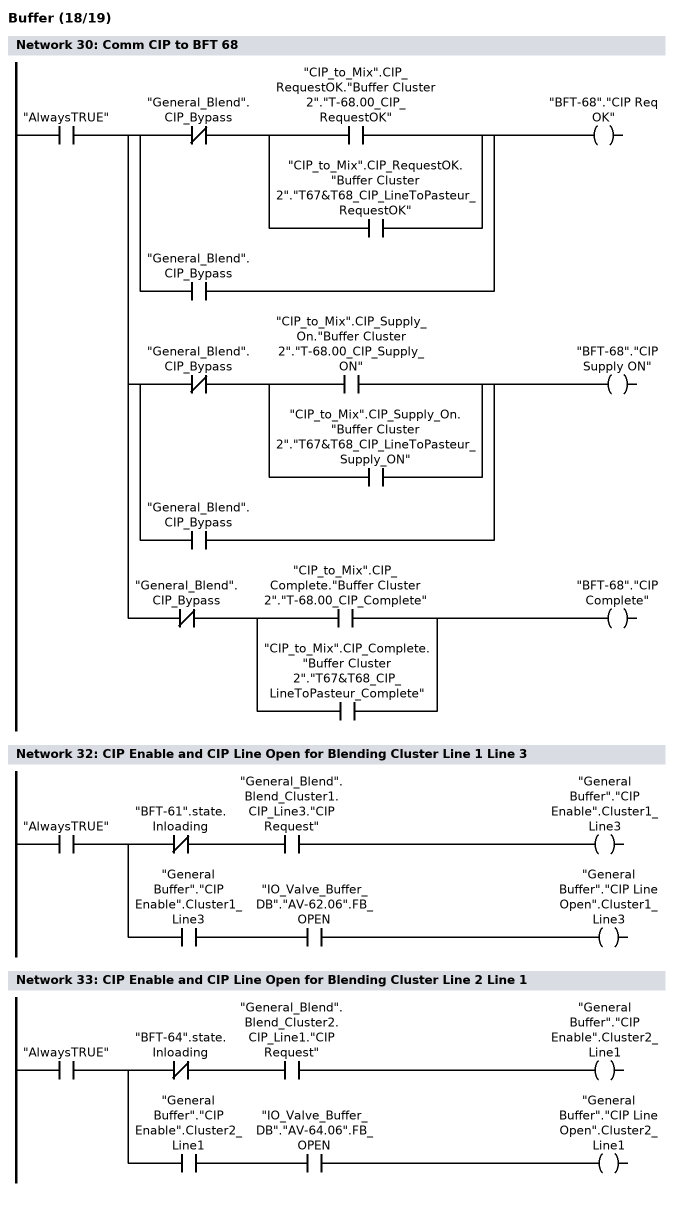
   RUNG wire#powerrail
      Contact( "AlwaysTRUE" )
      wire#w1
      I_Contact( "General_Blend".CIP_Bypass )
      wire#w2
      Contact( "CIP_to_Mix".CIP_RequestOK."Buffer Cluster 2"."T-68.00_CIP_RequestOK" )
      wire#w3
      Coil( "BFT-68"."CIP Req OK" )
   END_RUNG
   RUNG wire#w2
      Contact( "CIP_to_Mix".CIP_RequestOK."Buffer Cluster 2"."T67&T68_CIP_LineToPasteur_RequestOK" )
   END_RUNG wire#w3
   RUNG wire#w1
      Contact( "General_Blend".CIP_Bypass )
   END_RUNG wire#w3
   RUNG wire#w1
      I_Contact( "General_Blend".CIP_Bypass )
      wire#w4
      Contact( "CIP_to_Mix".CIP_Supply_On."Buffer Cluster 2"."T-68.00_CIP_Supply_ON" )
      wire#w5
      Coil( "BFT-68"."CIP Supply ON" )
   END_RUNG
   RUNG wire#w4
      Contact( "CIP_to_Mix".CIP_Supply_On."Buffer Cluster 2"."T67&T68_CIP_LineToPasteur_Supply_ON" )
   END_RUNG wire#w5
   RUNG wire#w1
      Contact( "General_Blend".CIP_Bypass )
   END_RUNG wire#w5
   RUNG wire#w1
      I_Contact( "General_Blend".CIP_Bypass )
      wire#w6
      Contact( "CIP_to_Mix".CIP_Complete."Buffer Cluster 2"."T-68.00_CIP_Complete" )
      wire#w7
      Coil( "BFT-68"."CIP Complete" )
   END_RUNG
   RUNG wire#w6
      Contact( "CIP_to_Mix".CIP_Complete."Buffer Cluster 2"."T67&T68_CIP_LineToPasteur_Complete" )
   END_RUNG wire#w7
   // the same network as SCL:
   "BFT-68"."CIP Req OK" := "AlwaysTRUE" AND ((NOT "General_Blend".CIP_Bypass AND ("CIP_to_Mix".CIP_RequestOK."Buffer Cluster 2"."T-68.00_CIP_RequestOK" OR "CIP_to_Mix".CIP_RequestOK."Buffer Cluster 2"."T67&T68_CIP_LineToPasteur_RequestOK")) OR "General_Blend".CIP_Bypass);
   "BFT-68"."CIP Supply ON" := "AlwaysTRUE" AND ((NOT "General_Blend".CIP_Bypass AND ("CIP_to_Mix".CIP_Supply_On."Buffer Cluster 2"."T-68.00_CIP_Supply_ON" OR "CIP_to_Mix".CIP_Supply_On."Buffer Cluster 2"."T67&T68_CIP_LineToPasteur_Supply_ON")) OR "General_Blend".CIP_Bypass);
   "BFT-68"."CIP Complete" := "AlwaysTRUE" AND NOT "General_Blend".CIP_Bypass AND ("CIP_to_Mix".CIP_Complete."Buffer Cluster 2"."T-68.00_CIP_Complete" OR "CIP_to_Mix".CIP_Complete."Buffer Cluster 2"."T67&T68_CIP_LineToPasteur_Complete");
END_REGION

REGION Network 32: CIP Enable and CIP Line Open for Blending Cluster Line 1 Line 3
   RUNG wire#powerrail
      Contact( "AlwaysTRUE" )
      wire#w1
      I_Contact( "BFT-61".state.Inloading )
      Contact( "General_Blend".Blend_Cluster1.CIP_Line3."CIP Request" )
      Coil( "General Buffer"."CIP Enable".Cluster1_Line3 )
   END_RUNG
   RUNG wire#w1
      Contact( "General Buffer"."CIP Enable".Cluster1_Line3 )
      Contact( "IO_Valve_Buffer_DB"."AV-62.06".FB_OPEN )
      Coil( "General Buffer"."CIP Line Open".Cluster1_Line3 )
   END_RUNG
   // the same network as SCL:
   "General Buffer"."CIP Enable".Cluster1_Line3 := "AlwaysTRUE" AND NOT "BFT-61".state.Inloading AND "General_Blend".Blend_Cluster1.CIP_Line3."CIP Request";
   "General Buffer"."CIP Line Open".Cluster1_Line3 := "AlwaysTRUE" AND "General Buffer"."CIP Enable".Cluster1_Line3 AND "IO_Valve_Buffer_DB"."AV-62.06".FB_OPEN;
END_REGION

REGION Network 33: CIP Enable and CIP Line Open for Blending Cluster Line 2 Line 1
   RUNG wire#powerrail
      Contact( "AlwaysTRUE" )
      wire#w1
      I_Contact( "BFT-64".state.Inloading )
      Contact( "General_Blend".Blend_Cluster2.CIP_Line1."CIP Request" )
      Coil( "General Buffer"."CIP Enable".Cluster2_Line1 )
   END_RUNG
   RUNG wire#w1
      Contact( "General Buffer"."CIP Enable".Cluster2_Line1 )
      Contact( "IO_Valve_Buffer_DB"."AV-64.06".FB_OPEN )
      Coil( "General Buffer"."CIP Line Open".Cluster2_Line1 )
   END_RUNG
   // the same network as SCL:
   "General Buffer"."CIP Enable".Cluster2_Line1 := "AlwaysTRUE" AND NOT "BFT-64".state.Inloading AND "General_Blend".Blend_Cluster2.CIP_Line1."CIP Request";
   "General Buffer"."CIP Line Open".Cluster2_Line1 := "AlwaysTRUE" AND "General Buffer"."CIP Enable".Cluster2_Line1 AND "IO_Valve_Buffer_DB"."AV-64.06".FB_OPEN;
END_REGION

REGION Network 34: CIP Enable and CIP Line Open for Blending Cluster Line 2 Line 2
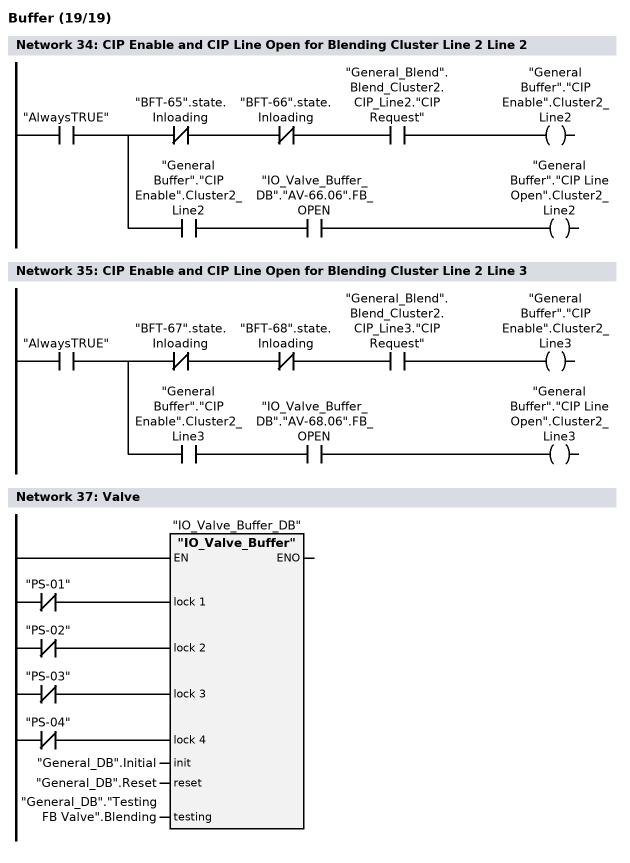
   RUNG wire#powerrail
      Contact( "AlwaysTRUE" )
      wire#w1
      I_Contact( "BFT-65".state.Inloading )
      I_Contact( "BFT-66".state.Inloading )
      Contact( "General_Blend".Blend_Cluster2.CIP_Line2."CIP Request" )
      Coil( "General Buffer"."CIP Enable".Cluster2_Line2 )
   END_RUNG
   RUNG wire#w1
      Contact( "General Buffer"."CIP Enable".Cluster2_Line2 )
      Contact( "IO_Valve_Buffer_DB"."AV-66.06".FB_OPEN )
      Coil( "General Buffer"."CIP Line Open".Cluster2_Line2 )
   END_RUNG
   // the same network as SCL:
   "General Buffer"."CIP Enable".Cluster2_Line2 := "AlwaysTRUE" AND NOT "BFT-65".state.Inloading AND NOT "BFT-66".state.Inloading AND "General_Blend".Blend_Cluster2.CIP_Line2."CIP Request";
   "General Buffer"."CIP Line Open".Cluster2_Line2 := "AlwaysTRUE" AND "General Buffer"."CIP Enable".Cluster2_Line2 AND "IO_Valve_Buffer_DB"."AV-66.06".FB_OPEN;
END_REGION

REGION Network 35: CIP Enable and CIP Line Open for Blending Cluster Line 2 Line 3
   RUNG wire#powerrail
      Contact( "AlwaysTRUE" )
      wire#w1
      I_Contact( "BFT-67".state.Inloading )
      I_Contact( "BFT-68".state.Inloading )
      Contact( "General_Blend".Blend_Cluster2.CIP_Line3."CIP Request" )
      Coil( "General Buffer"."CIP Enable".Cluster2_Line3 )
   END_RUNG
   RUNG wire#w1
      Contact( "General Buffer"."CIP Enable".Cluster2_Line3 )
      Contact( "IO_Valve_Buffer_DB"."AV-68.06".FB_OPEN )
      Coil( "General Buffer"."CIP Line Open".Cluster2_Line3 )
   END_RUNG
   // the same network as SCL:
   "General Buffer"."CIP Enable".Cluster2_Line3 := "AlwaysTRUE" AND NOT "BFT-67".state.Inloading AND NOT "BFT-68".state.Inloading AND "General_Blend".Blend_Cluster2.CIP_Line3."CIP Request";
   "General Buffer"."CIP Line Open".Cluster2_Line3 := "AlwaysTRUE" AND "General Buffer"."CIP Enable".Cluster2_Line3 AND "IO_Valve_Buffer_DB"."AV-68.06".FB_OPEN;
END_REGION

REGION Network 37: Valve
   RUNG wire#powerrail
      "IO_Valve_Buffer_DB"("lock 1" := wire#w1, "lock 2" := wire#w2, "lock 3" := wire#w3, "lock 4" := wire#w4, init := "General_DB".Initial, reset := "General_DB".Reset, testing := "General_DB"."Testing FB Valve".Blending)
   END_RUNG
   RUNG wire#powerrail
      I_Contact( "PS-01" )
   END_RUNG wire#w1
   RUNG wire#powerrail
      I_Contact( "PS-02" )
   END_RUNG wire#w2
   RUNG wire#powerrail
      I_Contact( "PS-03" )
   END_RUNG wire#w3
   RUNG wire#powerrail
      I_Contact( "PS-04" )
   END_RUNG wire#w4
   // the same network as SCL:
   "IO_Valve_Buffer_DB"("lock 1" := NOT "PS-01",   // "IO_Valve_Buffer"
                        "lock 2" := NOT "PS-02",
                        "lock 3" := NOT "PS-03",
                        "lock 4" := NOT "PS-04",
                        init := "General_DB".Initial,
                        reset := "General_DB".Reset,
                        testing := "General_DB"."Testing FB Valve".Blending);
END_REGION
END_FUNCTION

FUNCTION_BLOCK "Buffer_Tank"   // FB110, LAD
{ S7_Optimized_Access := 'TRUE' }
VERSION : 0.1
// stored: AutoNumber false, IsIECCheckEnabled false, IsRetainMemResEnabled false, MemoryReserve 100, SetENOAutomatically false, UDAEnableTagReadback false
   VAR_INPUT
      IN_LT01 : Real;
      "Tank w Circulation" : Bool;
      AlarmProd_pasteur : Bool;
      HighLevel_pasteur : Bool;
      IN_FBAV_Inload : Bool;
      IN_FBAV_CIP_Tank : Bool;
      IN_FBAV_CIP_Line : Bool;
      IN_FBAV_Outlet : Bool;
      IN_FBAV_Transfer : Bool;
      IN_FBP_Transfer : Bool;
      IN_FBXA : Bool;
      IN_FBP_Circulation : Bool;
      IN_Product_Ready : Bool;
      IN_Product_TransferOnProg : Bool;
      "Inload Busy" : Bool;
      "CIP Pulse" : Bool;
      "CIP Req OK" : Bool;
      "CIP Supply ON" : Bool;
      "CIP In Progress" : Bool;
      "CIP Complete" : Bool;
      "CIP Busy" : Bool;
   END_VAR
   VAR_OUTPUT
      Out_AV_Inload : Bool;
      Out_AV_Drain_In : Bool;
      Out_AV_CIP_Tank : Bool;
      Out_AV_CIP_Line : Bool;
      Out_AV_Outlet : Bool;
      Out_AV_Transfer : Bool;
      Out_P_Transfer : Bool;
      Out_P_Transfer_SP : Real;
      Out_XA : Bool;
      Out_XA_SP : Real;
      Out_P_Circulation : Bool;
      Out_Prod_Req : Bool;
      Out_Prod_LineOpen : Bool;
      Out_CIP_Tank_Req : Bool;
      Out_CIP_Line_Req : Bool;
      Out_CIP_Tank_LineOpen : Bool;
      Out_CIP_Line_LineOpen : Bool;
   END_VAR
   VAR
      cmd : Struct
         Inload : Bool;
         Drain_In : Bool;
         Ready_for_Transfer : Bool;
         CIP_Tank : Bool;
         CIP_Line : Bool;
         Agitator_Mode : Bool;
         Agitator_Man_OnOff : Bool;
         Agitator_SpeedMode : Bool;
         Circulation : Bool;
      END_STRUCT;
   END_VAR
   VAR RETAIN
      param : Struct
         L_Lo_Lim : Real;
         L_Hi_Lim : Real := 100.0;
         L_Hys : Real := 2.0;
         "Circulation Level" : Real := 20.0;
         SP_Level_HL : Real := 100.0;
         SP_Level_ML : Real := 80.0;
         SP_Level_LL : Real := 10.0;
         DrainIn : DInt := 10;
         SP_Pump_Transfer : Real := 80.0;
         SP_Pump_CIP : Real := 80.0;
         SP_Agitator : Real := 50.0;
         SP_Level_Agi_ON1 : Real := 20.0;
         SP_Level_Agi_OFF1 : Real := 49.0;
         SP_Level_Agi_ON2 : Real := 50.0;
         SP_Level_Agi_OFF2 : Real := 64.0;
         SP_Level_Agi_ON3 : Real := 65.0;
         "CIP Ret On" : Real := 5.0;
         "CIP Ret Off" : Real;
      END_STRUCT;
   END_VAR
   VAR
      state : Struct
         "Tank LL" : Bool;
         "Tank ML" : Bool;
         "Tank HL" : Bool;
         "Tank CIP En" : Bool;
         "Tank CIP" : Bool;
         "Line CIP En" : Bool;
         "Line CIP" : Bool;
         "Ready for Transfer En" : Bool;
         "Ready for Transfer" : Bool;
         Inloading : Bool;
         "Inload En" : Bool;
         L_Agi_ON1 : Bool;
         L_Agi_ON2 : Bool;
         L_Agi_ON3 : Bool;
         Tank_Circulation : Bool;
         "Circulation Enable" : Bool;
         Circulation : Bool;
         "Transfer on Prog" : Bool;
         "CIP Return On" : Bool;
         "CIP Req" : Bool;
      END_STRUCT;
      alwaysOn : Bool;
      L_Hys_Abs : Real;
      Hys_Level_LL : Real;
      Hys_Level_ML : Real;
      Hys_Level_HL : Real;
      Hys_Level_Circ : Real;
   END_VAR
   VAR DB_SPECIFIC
      r : Struct
         PosE1 : Bool;
         PosE2 : Bool;
         PosE3 : Bool;
         PosE4 : Bool;
         PosE5 : Bool;
         PosE6 : Bool;
         PosE7 : Bool;
         PosE8 : Bool;
         PosE9 : Bool;
         PosE10 : Bool;
         PosE11 : Bool;
         PosE12 : Bool;
         PosE13 : Bool;
         PosE14 : Bool;
         PosE15 : Bool;
         PosE16 : Bool;
         PosE17 : Bool;
         PosE18 : Bool;
         PosE19 : Bool;
         PosE20 : Bool;
         PosE21 : Bool;
         PosE22 : Bool;
         PosE23 : Bool;
         PosE24 : Bool;
         PosE25 : Bool;
         PosE26 : Bool;
         PosE27 : Bool;
         PosE28 : Bool;
         PosE29 : Bool;
         PosE30 : Bool;
         PosE31 : Bool;
         PosE32 : Bool;
      END_STRUCT;
      Actuator : Struct
         AV_Inload : Bool;
         AV_Drain_In : Bool;
         AV_Outlet : Bool;
         AV_Transfer : Bool;
         AV_CIP_Tank : Bool;
         AV_CIP_Line : Bool;
         P_Transfer : Bool;
         P_CIP : Bool;
         Agitator_level : Bool;
      END_STRUCT;
   END_VAR
   VAR
      DrainIn_OnTime : TON_TIME;
      DrainIn_OffTime : TOF_TIME;
      InloadAV_OffTime : TOF_TIME;
      DrainIn_MS : DInt;
      L_AgiTim : TON_TIME;
   END_VAR
   VAR_TEMP   // added for the SCL form of the ladder/FBD networks
      _w1 : Bool;
      _w2 : Bool;
      _w3 : Bool;
   END_VAR
BEGIN

REGION Network 1: always On
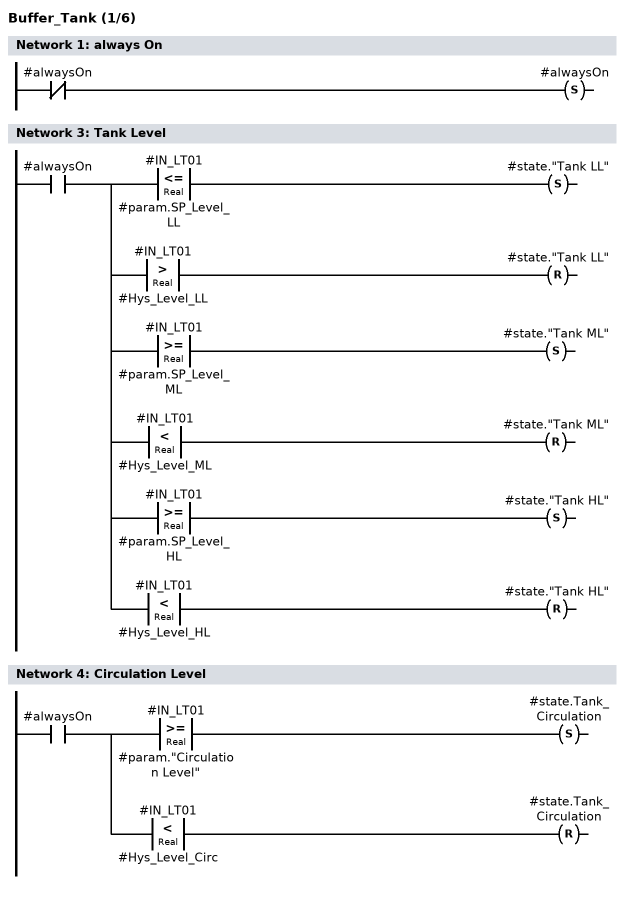
   RUNG wire#powerrail
      I_Contact( #alwaysOn )
      S_Coil( #alwaysOn )
   END_RUNG
   // the same network as SCL:
   IF NOT #alwaysOn THEN #alwaysOn := TRUE; END_IF;
END_REGION

NETWORK
TITLE = Hys Calculation
//Level Hys Absolute
      L     #param.L_Hi_Lim;
      L     #param.L_Lo_Lim;
      -R;
      L     100.0;
      /R;
      L     #param.L_Hys;
      *R;
      T     #L_Hys_Abs;
//Tank High Level
      L     #param.SP_Level_HL;
      L     #L_Hys_Abs;
      -R;
      T     #Hys_Level_HL;
//Tank Mid Level
      L     #param.SP_Level_ML;
      L     #L_Hys_Abs;
      -R;
      T     #Hys_Level_ML;
//Tank Low Level
      L     #param.SP_Level_LL;
      L     #L_Hys_Abs;
      +R;
      T     #Hys_Level_LL;
//Level Circulation
      L     #param."Circulation Level";
      L     #L_Hys_Abs;
      -R;
      T     #Hys_Level_Circ;



REGION Network 3: Tank Level
   RUNG wire#powerrail
      Contact( #alwaysOn )
      wire#w1
      { S7_Templates := "SrcType := Real" } LE_Contact(in1 := #IN_LT01, in2 := #param.SP_Level_LL)
      S_Coil( #state."Tank LL" )
   END_RUNG
   RUNG wire#w1
      { S7_Templates := "SrcType := Real" } GT_Contact(in1 := #IN_LT01, in2 := #Hys_Level_LL)
      R_Coil( #state."Tank LL" )
   END_RUNG
   RUNG wire#w1
      { S7_Templates := "SrcType := Real" } GE_Contact(in1 := #IN_LT01, in2 := #param.SP_Level_ML)
      S_Coil( #state."Tank ML" )
   END_RUNG
   RUNG wire#w1
      { S7_Templates := "SrcType := Real" } LT_Contact(in1 := #IN_LT01, in2 := #Hys_Level_ML)
      R_Coil( #state."Tank ML" )
   END_RUNG
   RUNG wire#w1
      { S7_Templates := "SrcType := Real" } GE_Contact(in1 := #IN_LT01, in2 := #param.SP_Level_HL)
      S_Coil( #state."Tank HL" )
   END_RUNG
   RUNG wire#w1
      { S7_Templates := "SrcType := Real" } LT_Contact(in1 := #IN_LT01, in2 := #Hys_Level_HL)
      R_Coil( #state."Tank HL" )
   END_RUNG
   // the same network as SCL:
   IF #alwaysOn AND (#IN_LT01 <= #param.SP_Level_LL) THEN #state."Tank LL" := TRUE; END_IF;
   IF #alwaysOn AND (#IN_LT01 > #Hys_Level_LL) THEN #state."Tank LL" := FALSE; END_IF;
   IF #alwaysOn AND (#IN_LT01 >= #param.SP_Level_ML) THEN #state."Tank ML" := TRUE; END_IF;
   IF #alwaysOn AND (#IN_LT01 < #Hys_Level_ML) THEN #state."Tank ML" := FALSE; END_IF;
   IF #alwaysOn AND (#IN_LT01 >= #param.SP_Level_HL) THEN #state."Tank HL" := TRUE; END_IF;
   IF #alwaysOn AND (#IN_LT01 < #Hys_Level_HL) THEN #state."Tank HL" := FALSE; END_IF;
END_REGION

REGION Network 4: Circulation Level
   RUNG wire#powerrail
      Contact( #alwaysOn )
      wire#w1
      { S7_Templates := "SrcType := Real" } GE_Contact(in1 := #IN_LT01, in2 := #param."Circulation Level")
      S_Coil( #state.Tank_Circulation )
   END_RUNG
   RUNG wire#w1
      { S7_Templates := "SrcType := Real" } LT_Contact(in1 := #IN_LT01, in2 := #Hys_Level_Circ)
      R_Coil( #state.Tank_Circulation )
   END_RUNG
   // the same network as SCL:
   IF #alwaysOn AND (#IN_LT01 >= #param."Circulation Level") THEN #state.Tank_Circulation := TRUE; END_IF;
   IF #alwaysOn AND (#IN_LT01 < #Hys_Level_Circ) THEN #state.Tank_Circulation := FALSE; END_IF;
END_REGION

REGION Network 5: Agitator Level ON-OFF
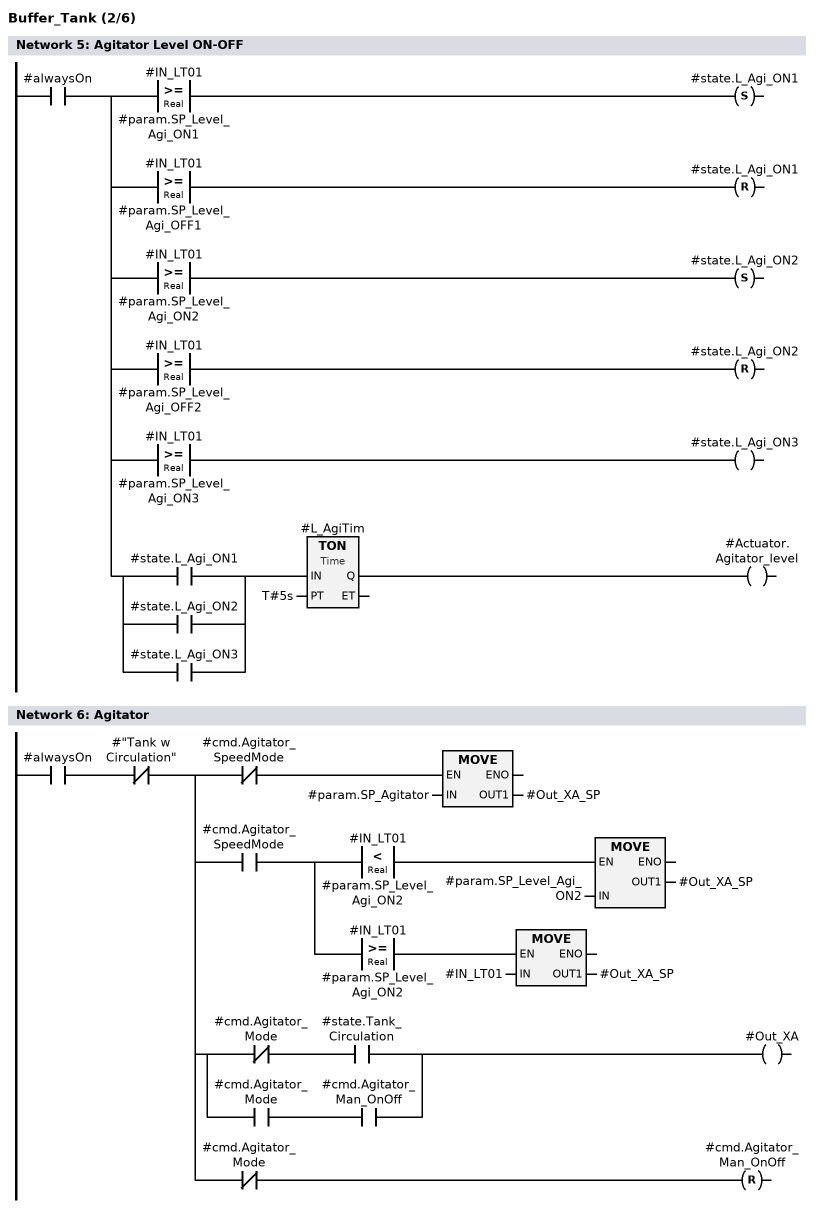
   RUNG wire#powerrail
      Contact( #alwaysOn )
      wire#w1
      { S7_Templates := "SrcType := Real" } GE_Contact(in1 := #IN_LT01, in2 := #param.SP_Level_Agi_ON1)
      S_Coil( #state.L_Agi_ON1 )
   END_RUNG
   RUNG wire#w1
      { S7_Templates := "SrcType := Real" } GE_Contact(in1 := #IN_LT01, in2 := #param.SP_Level_Agi_OFF1)
      R_Coil( #state.L_Agi_ON1 )
   END_RUNG
   RUNG wire#w1
      { S7_Templates := "SrcType := Real" } GE_Contact(in1 := #IN_LT01, in2 := #param.SP_Level_Agi_ON2)
      S_Coil( #state.L_Agi_ON2 )
   END_RUNG
   RUNG wire#w1
      { S7_Templates := "SrcType := Real" } GE_Contact(in1 := #IN_LT01, in2 := #param.SP_Level_Agi_OFF2)
      R_Coil( #state.L_Agi_ON2 )
   END_RUNG
   RUNG wire#w1
      { S7_Templates := "SrcType := Real" } GE_Contact(in1 := #IN_LT01, in2 := #param.SP_Level_Agi_ON3)
      Coil( #state.L_Agi_ON3 )
   END_RUNG
   RUNG wire#w1
      Contact( #state.L_Agi_ON1 )
      wire#w2
      { S7_Templates := "time_type := Time" } #L_AgiTim.TON(pt := T#5s, et =>)
      Coil( #Actuator.Agitator_level )
   END_RUNG
   RUNG wire#w1
      Contact( #state.L_Agi_ON2 )
   END_RUNG wire#w2
   RUNG wire#w1
      Contact( #state.L_Agi_ON3 )
   END_RUNG wire#w2
   // the same network as SCL:
   IF #alwaysOn AND (#IN_LT01 >= #param.SP_Level_Agi_ON1) THEN #state.L_Agi_ON1 := TRUE; END_IF;
   IF #alwaysOn AND (#IN_LT01 >= #param.SP_Level_Agi_OFF1) THEN #state.L_Agi_ON1 := FALSE; END_IF;
   IF #alwaysOn AND (#IN_LT01 >= #param.SP_Level_Agi_ON2) THEN #state.L_Agi_ON2 := TRUE; END_IF;
   IF #alwaysOn AND (#IN_LT01 >= #param.SP_Level_Agi_OFF2) THEN #state.L_Agi_ON2 := FALSE; END_IF;
   #state.L_Agi_ON3 := #alwaysOn AND (#IN_LT01 >= #param.SP_Level_Agi_ON3);
   #L_AgiTim(IN := #alwaysOn AND (#state.L_Agi_ON1 OR #state.L_Agi_ON2 OR #state.L_Agi_ON3), PT := T#5s);   // TON
   #Actuator.Agitator_level := #L_AgiTim.Q;
END_REGION

REGION Network 6: Agitator
   RUNG wire#powerrail
      Contact( #alwaysOn )
      I_Contact( #"Tank w Circulation" )
      wire#w1
      I_Contact( #cmd.Agitator_SpeedMode )
      Move(in := #param.SP_Agitator, out1 => #Out_XA_SP)
   END_RUNG
   RUNG wire#w1
      Contact( #cmd.Agitator_SpeedMode )
      wire#w2
      { S7_Templates := "SrcType := Real" } LT_Contact(in1 := #IN_LT01, in2 := #param.SP_Level_Agi_ON2)
      Move(in := #param.SP_Level_Agi_ON2, out1 => #Out_XA_SP)
   END_RUNG
   RUNG wire#w2
      { S7_Templates := "SrcType := Real" } GE_Contact(in1 := #IN_LT01, in2 := #param.SP_Level_Agi_ON2)
      Move(in := #IN_LT01, out1 => #Out_XA_SP)
   END_RUNG
   RUNG wire#w1
      I_Contact( #cmd.Agitator_Mode )
      Contact( #state.Tank_Circulation )
      wire#w3
      Coil( #Out_XA )
   END_RUNG
   RUNG wire#w1
      Contact( #cmd.Agitator_Mode )
      Contact( #cmd.Agitator_Man_OnOff )
   END_RUNG wire#w3
   RUNG wire#w1
      I_Contact( #cmd.Agitator_Mode )
      R_Coil( #cmd.Agitator_Man_OnOff )
   END_RUNG
   // the same network as SCL:
   #_w1 := #alwaysOn AND NOT #"Tank w Circulation";
   IF #_w1 AND NOT #cmd.Agitator_SpeedMode THEN #Out_XA_SP := #param.SP_Agitator; END_IF;
   #_w2 := #_w1 AND #cmd.Agitator_SpeedMode;
   IF #_w2 AND (#IN_LT01 < #param.SP_Level_Agi_ON2) THEN #Out_XA_SP := #param.SP_Level_Agi_ON2; END_IF;
   IF #_w2 AND (#IN_LT01 >= #param.SP_Level_Agi_ON2) THEN #Out_XA_SP := #IN_LT01; END_IF;
   #Out_XA := #_w1 AND ((NOT #cmd.Agitator_Mode AND #state.Tank_Circulation) OR (#cmd.Agitator_Mode AND #cmd.Agitator_Man_OnOff));
   IF #_w1 AND NOT #cmd.Agitator_Mode THEN #cmd.Agitator_Man_OnOff := FALSE; END_IF;
END_REGION

REGION Network 7: Circulation
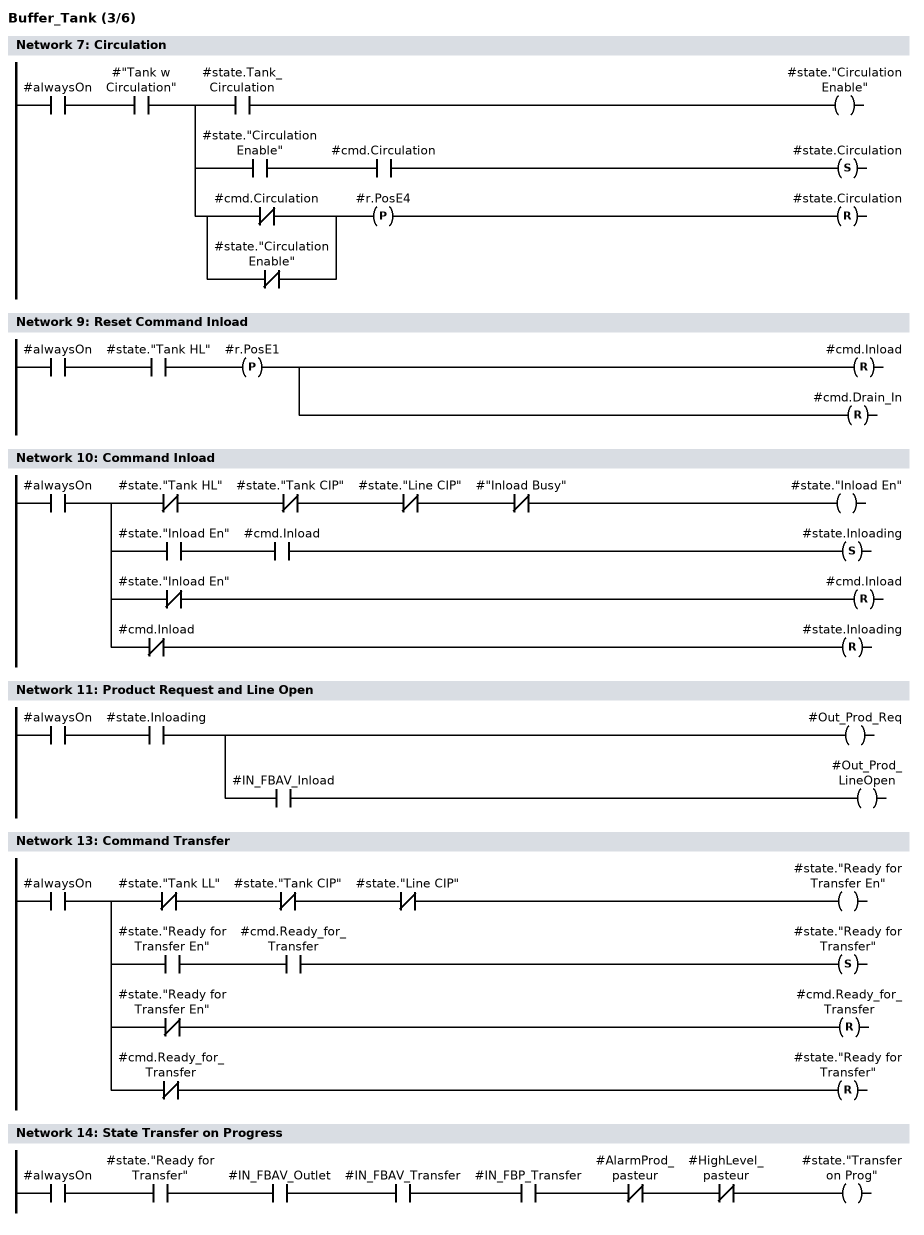
   RUNG wire#powerrail
      Contact( #alwaysOn )
      Contact( #"Tank w Circulation" )
      wire#w1
      Contact( #state.Tank_Circulation )
      Coil( #state."Circulation Enable" )
   END_RUNG
   RUNG wire#w1
      Contact( #state."Circulation Enable" )
      Contact( #cmd.Circulation )
      S_Coil( #state.Circulation )
   END_RUNG
   RUNG wire#w1
      I_Contact( #cmd.Circulation )
      wire#w2
      P_Trig( #r.PosE4 )
      R_Coil( #state.Circulation )
   END_RUNG
   RUNG wire#w1
      I_Contact( #state."Circulation Enable" )
   END_RUNG wire#w2
   // the same network as SCL:
   #_w1 := #alwaysOn AND #"Tank w Circulation";
   #state."Circulation Enable" := #_w1 AND #state.Tank_Circulation;
   IF #_w1 AND #state."Circulation Enable" AND #cmd.Circulation THEN #state.Circulation := TRUE; END_IF;
   #_w2 := #_w1 AND (NOT #cmd.Circulation OR NOT #state."Circulation Enable");
   #_w3 := #_w2 AND NOT #r.PosE4;   // rising edge
   #r.PosE4 := #_w2;
   IF #_w3 THEN #state.Circulation := FALSE; END_IF;
END_REGION

REGION Network 9: Reset Command Inload
   RUNG wire#powerrail
      Contact( #alwaysOn )
      Contact( #state."Tank HL" )
      P_Trig( #r.PosE1 )
      wire#w1
      R_Coil( #cmd.Inload )
   END_RUNG
   RUNG wire#w1
      R_Coil( #cmd.Drain_In )
   END_RUNG
   // the same network as SCL:
   #_w1 := #alwaysOn AND #state."Tank HL";
   #_w2 := #_w1 AND NOT #r.PosE1;   // rising edge
   #r.PosE1 := #_w1;
   IF #_w2 THEN
       #cmd.Inload := FALSE;
       #cmd.Drain_In := FALSE;
   END_IF;
END_REGION

REGION Network 10: Command Inload
   RUNG wire#powerrail
      Contact( #alwaysOn )
      wire#w1
      I_Contact( #state."Tank HL" )
      I_Contact( #state."Tank CIP" )
      I_Contact( #state."Line CIP" )
      I_Contact( #"Inload Busy" )
      Coil( #state."Inload En" )
   END_RUNG
   RUNG wire#w1
      Contact( #state."Inload En" )
      Contact( #cmd.Inload )
      S_Coil( #state.Inloading )
   END_RUNG
   RUNG wire#w1
      I_Contact( #state."Inload En" )
      R_Coil( #cmd.Inload )
   END_RUNG
   RUNG wire#w1
      I_Contact( #cmd.Inload )
      R_Coil( #state.Inloading )
   END_RUNG
   // the same network as SCL:
   #state."Inload En" := #alwaysOn AND NOT #state."Tank HL" AND NOT #state."Tank CIP" AND NOT #state."Line CIP" AND NOT #"Inload Busy";
   IF #alwaysOn AND #state."Inload En" AND #cmd.Inload THEN #state.Inloading := TRUE; END_IF;
   IF #alwaysOn AND NOT #state."Inload En" THEN #cmd.Inload := FALSE; END_IF;
   IF #alwaysOn AND NOT #cmd.Inload THEN #state.Inloading := FALSE; END_IF;
END_REGION

REGION Network 11: Product Request and Line Open
   RUNG wire#powerrail
      Contact( #alwaysOn )
      Contact( #state.Inloading )
      wire#w1
      Coil( #Out_Prod_Req )
   END_RUNG
   RUNG wire#w1
      Contact( #IN_FBAV_Inload )
      Coil( #Out_Prod_LineOpen )
   END_RUNG
   // the same network as SCL:
   #Out_Prod_Req := #alwaysOn AND #state.Inloading;
   #Out_Prod_LineOpen := #Out_Prod_Req AND #IN_FBAV_Inload;
END_REGION

REGION Network 13: Command Transfer
   RUNG wire#powerrail
      Contact( #alwaysOn )
      wire#w1
      I_Contact( #state."Tank LL" )
      I_Contact( #state."Tank CIP" )
      I_Contact( #state."Line CIP" )
      Coil( #state."Ready for Transfer En" )
   END_RUNG
   RUNG wire#w1
      Contact( #state."Ready for Transfer En" )
      Contact( #cmd.Ready_for_Transfer )
      S_Coil( #state."Ready for Transfer" )
   END_RUNG
   RUNG wire#w1
      I_Contact( #state."Ready for Transfer En" )
      R_Coil( #cmd.Ready_for_Transfer )
   END_RUNG
   RUNG wire#w1
      I_Contact( #cmd.Ready_for_Transfer )
      R_Coil( #state."Ready for Transfer" )
   END_RUNG
   // the same network as SCL:
   #state."Ready for Transfer En" := #alwaysOn AND NOT #state."Tank LL" AND NOT #state."Tank CIP" AND NOT #state."Line CIP";
   IF #alwaysOn AND #state."Ready for Transfer En" AND #cmd.Ready_for_Transfer THEN
       #state."Ready for Transfer" := TRUE;
   END_IF;
   IF #alwaysOn AND NOT #state."Ready for Transfer En" THEN #cmd.Ready_for_Transfer := FALSE; END_IF;
   IF #alwaysOn AND NOT #cmd.Ready_for_Transfer THEN #state."Ready for Transfer" := FALSE; END_IF;
END_REGION

REGION Network 14: State Transfer on Progress
   RUNG wire#powerrail
      Contact( #alwaysOn )
      Contact( #state."Ready for Transfer" )
      Contact( #IN_FBAV_Outlet )
      Contact( #IN_FBAV_Transfer )
      Contact( #IN_FBP_Transfer )
      I_Contact( #AlarmProd_pasteur )
      I_Contact( #HighLevel_pasteur )
      Coil( #state."Transfer on Prog" )
   END_RUNG
   // the same network as SCL:
   #state."Transfer on Prog" := #alwaysOn AND #state."Ready for Transfer" AND #IN_FBAV_Outlet AND #IN_FBAV_Transfer AND #IN_FBP_Transfer AND NOT #AlarmProd_pasteur AND NOT #HighLevel_pasteur;
END_REGION

REGION Network 16: Command CIP
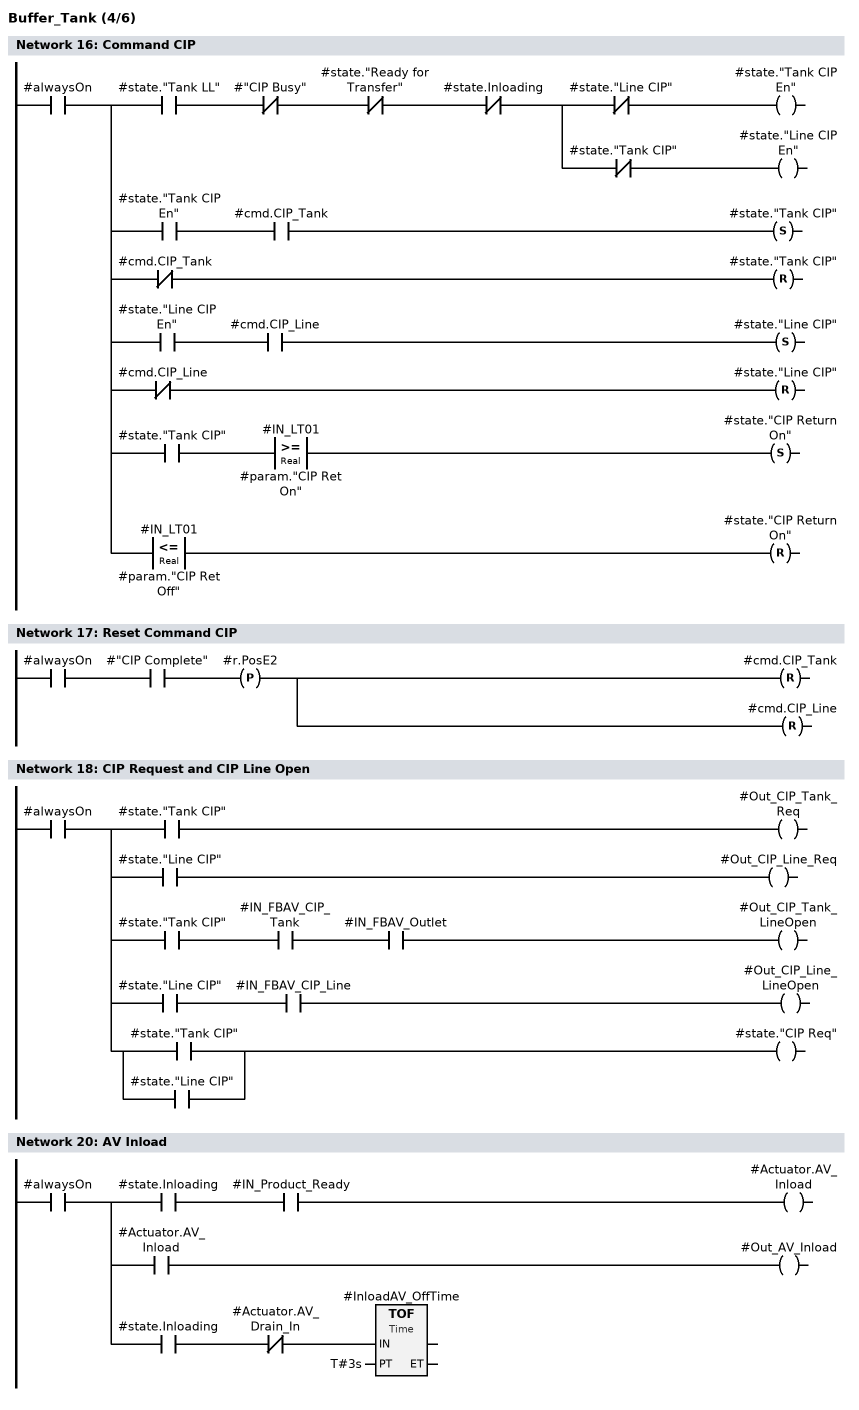
   RUNG wire#powerrail
      Contact( #alwaysOn )
      wire#w1
      Contact( #state."Tank LL" )
      I_Contact( #"CIP Busy" )
      I_Contact( #state."Ready for Transfer" )
      I_Contact( #state.Inloading )
      wire#w2
      I_Contact( #state."Line CIP" )
      Coil( #state."Tank CIP En" )
   END_RUNG
   RUNG wire#w2
      I_Contact( #state."Tank CIP" )
      Coil( #state."Line CIP En" )
   END_RUNG
   RUNG wire#w1
      Contact( #state."Tank CIP En" )
      Contact( #cmd.CIP_Tank )
      S_Coil( #state."Tank CIP" )
   END_RUNG
   RUNG wire#w1
      I_Contact( #cmd.CIP_Tank )
      R_Coil( #state."Tank CIP" )
   END_RUNG
   RUNG wire#w1
      Contact( #state."Line CIP En" )
      Contact( #cmd.CIP_Line )
      S_Coil( #state."Line CIP" )
   END_RUNG
   RUNG wire#w1
      I_Contact( #cmd.CIP_Line )
      R_Coil( #state."Line CIP" )
   END_RUNG
   RUNG wire#w1
      Contact( #state."Tank CIP" )
      { S7_Templates := "SrcType := Real" } GE_Contact(in1 := #IN_LT01, in2 := #param."CIP Ret On")
      S_Coil( #state."CIP Return On" )
   END_RUNG
   RUNG wire#w1
      { S7_Templates := "SrcType := Real" } LE_Contact(in1 := #IN_LT01, in2 := #param."CIP Ret Off")
      R_Coil( #state."CIP Return On" )
   END_RUNG
   // the same network as SCL:
   #_w1 := #alwaysOn AND #state."Tank LL" AND NOT #"CIP Busy" AND NOT #state."Ready for Transfer" AND NOT #state.Inloading;
   #state."Tank CIP En" := #_w1 AND NOT #state."Line CIP";
   #state."Line CIP En" := #_w1 AND NOT #state."Tank CIP";
   IF #alwaysOn AND #state."Tank CIP En" AND #cmd.CIP_Tank THEN #state."Tank CIP" := TRUE; END_IF;
   IF #alwaysOn AND NOT #cmd.CIP_Tank THEN #state."Tank CIP" := FALSE; END_IF;
   IF #alwaysOn AND #state."Line CIP En" AND #cmd.CIP_Line THEN #state."Line CIP" := TRUE; END_IF;
   IF #alwaysOn AND NOT #cmd.CIP_Line THEN #state."Line CIP" := FALSE; END_IF;
   IF #alwaysOn AND #state."Tank CIP" AND (#IN_LT01 >= #param."CIP Ret On") THEN
       #state."CIP Return On" := TRUE;
   END_IF;
   IF #alwaysOn AND (#IN_LT01 <= #param."CIP Ret Off") THEN #state."CIP Return On" := FALSE; END_IF;
END_REGION

REGION Network 17: Reset Command CIP
   RUNG wire#powerrail
      Contact( #alwaysOn )
      Contact( #"CIP Complete" )
      P_Trig( #r.PosE2 )
      wire#w1
      R_Coil( #cmd.CIP_Tank )
   END_RUNG
   RUNG wire#w1
      R_Coil( #cmd.CIP_Line )
   END_RUNG
   // the same network as SCL:
   #_w1 := #alwaysOn AND #"CIP Complete";
   #_w2 := #_w1 AND NOT #r.PosE2;   // rising edge
   #r.PosE2 := #_w1;
   IF #_w2 THEN
       #cmd.CIP_Tank := FALSE;
       #cmd.CIP_Line := FALSE;
   END_IF;
END_REGION

REGION Network 18: CIP Request and CIP Line Open
   RUNG wire#powerrail
      Contact( #alwaysOn )
      wire#w1
      Contact( #state."Tank CIP" )
      Coil( #Out_CIP_Tank_Req )
   END_RUNG
   RUNG wire#w1
      Contact( #state."Line CIP" )
      Coil( #Out_CIP_Line_Req )
   END_RUNG
   RUNG wire#w1
      Contact( #state."Tank CIP" )
      Contact( #IN_FBAV_CIP_Tank )
      Contact( #IN_FBAV_Outlet )
      Coil( #Out_CIP_Tank_LineOpen )
   END_RUNG
   RUNG wire#w1
      Contact( #state."Line CIP" )
      Contact( #IN_FBAV_CIP_Line )
      Coil( #Out_CIP_Line_LineOpen )
   END_RUNG
   RUNG wire#w1
      Contact( #state."Tank CIP" )
      wire#w2
      Coil( #state."CIP Req" )
   END_RUNG
   RUNG wire#w1
      Contact( #state."Line CIP" )
   END_RUNG wire#w2
   // the same network as SCL:
   #Out_CIP_Tank_Req := #alwaysOn AND #state."Tank CIP";
   #Out_CIP_Line_Req := #alwaysOn AND #state."Line CIP";
   #Out_CIP_Tank_LineOpen := #alwaysOn AND #state."Tank CIP" AND #IN_FBAV_CIP_Tank AND #IN_FBAV_Outlet;
   #Out_CIP_Line_LineOpen := #alwaysOn AND #state."Line CIP" AND #IN_FBAV_CIP_Line;
   #state."CIP Req" := #alwaysOn AND (#state."Tank CIP" OR #state."Line CIP");
END_REGION

REGION Network 20: AV Inload
   RUNG wire#powerrail
      Contact( #alwaysOn )
      wire#w1
      Contact( #state.Inloading )
      Contact( #IN_Product_Ready )
      Coil( #Actuator.AV_Inload )
   END_RUNG
   RUNG wire#w1
      Contact( #Actuator.AV_Inload )
      Coil( #Out_AV_Inload )
   END_RUNG
   RUNG wire#w1
      Contact( #state.Inloading )
      I_Contact( #Actuator.AV_Drain_In )
      { S7_Templates := "time_type := Time" } #InloadAV_OffTime.TOF(pt := T#3s, et =>)
   END_RUNG
   // the same network as SCL:
   #Actuator.AV_Inload := #alwaysOn AND #state.Inloading AND #IN_Product_Ready;
   #Out_AV_Inload := #alwaysOn AND #Actuator.AV_Inload;
   #InloadAV_OffTime(IN := #alwaysOn AND #state.Inloading AND NOT #Actuator.AV_Drain_In, PT := T#3s);   // TOF
END_REGION

REGION Network 21: AV Drain In
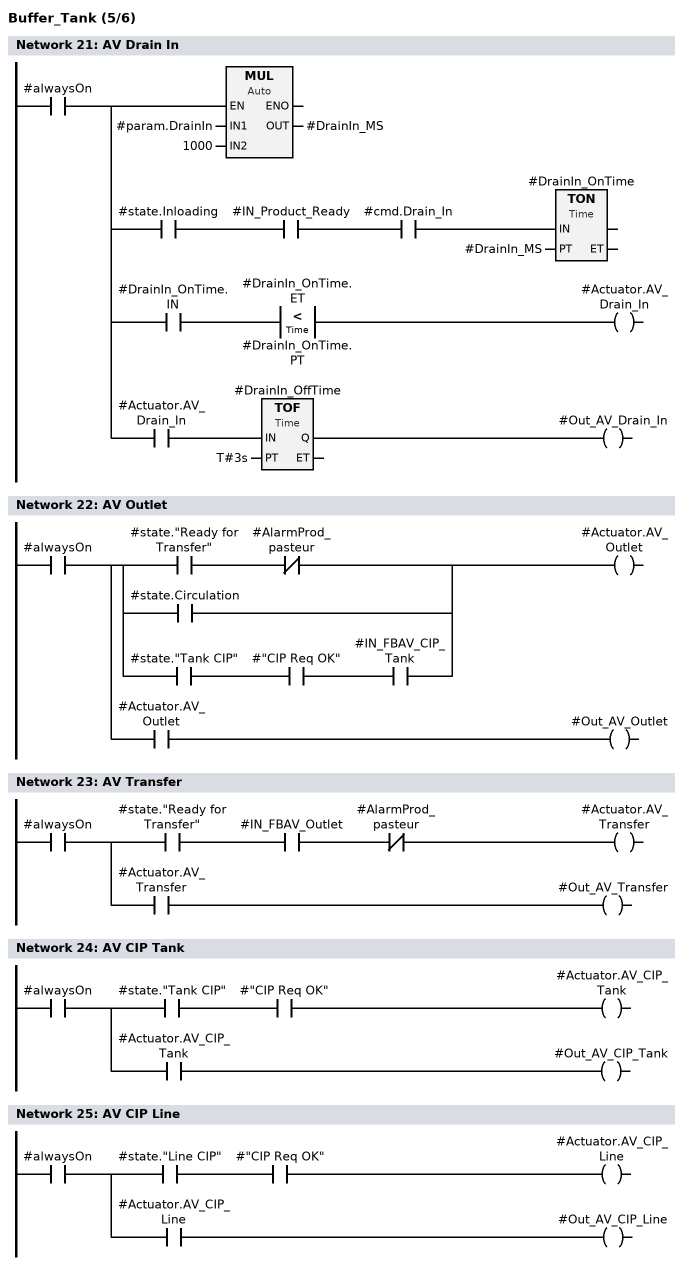
   RUNG wire#powerrail
      Contact( #alwaysOn )
      wire#w1
      Mul(in1 := #param.DrainIn, in2 := 1000, out => #DrainIn_MS)
   END_RUNG
   RUNG wire#w1
      Contact( #state.Inloading )
      Contact( #IN_Product_Ready )
      Contact( #cmd.Drain_In )
      { S7_Templates := "time_type := Time" } #DrainIn_OnTime.TON(pt := #DrainIn_MS, et =>)
   END_RUNG
   RUNG wire#w1
      Contact( #DrainIn_OnTime.IN )
      { S7_Templates := "SrcType := Time" } LT_Contact(in1 := #DrainIn_OnTime.ET, in2 := #DrainIn_OnTime.PT)
      Coil( #Actuator.AV_Drain_In )
   END_RUNG
   RUNG wire#w1
      Contact( #Actuator.AV_Drain_In )
      { S7_Templates := "time_type := Time" } #DrainIn_OffTime.TOF(pt := T#3s, et =>)
      Coil( #Out_AV_Drain_In )
   END_RUNG
   // the same network as SCL:
   IF #alwaysOn THEN #DrainIn_MS := #param.DrainIn * 1000; END_IF;
   #DrainIn_OnTime(IN := #alwaysOn AND #state.Inloading AND #IN_Product_Ready AND #cmd.Drain_In,   // TON
                   PT := #DrainIn_MS);
   #Actuator.AV_Drain_In := #alwaysOn AND #DrainIn_OnTime.IN AND (#DrainIn_OnTime.ET < #DrainIn_OnTime.PT);
   #DrainIn_OffTime(IN := #alwaysOn AND #Actuator.AV_Drain_In, PT := T#3s);   // TOF
   #Out_AV_Drain_In := #DrainIn_OffTime.Q;
END_REGION

REGION Network 22: AV Outlet
   RUNG wire#powerrail
      Contact( #alwaysOn )
      wire#w1
      Contact( #state."Ready for Transfer" )
      I_Contact( #AlarmProd_pasteur )
      wire#w2
      Coil( #Actuator.AV_Outlet )
   END_RUNG
   RUNG wire#w1
      Contact( #state.Circulation )
   END_RUNG wire#w2
   RUNG wire#w1
      Contact( #state."Tank CIP" )
      Contact( #"CIP Req OK" )
      Contact( #IN_FBAV_CIP_Tank )
   END_RUNG wire#w2
   RUNG wire#w1
      Contact( #Actuator.AV_Outlet )
      Coil( #Out_AV_Outlet )
   END_RUNG
   // the same network as SCL:
   #Actuator.AV_Outlet := #alwaysOn AND ((#state."Ready for Transfer" AND NOT #AlarmProd_pasteur) OR #state.Circulation OR (#state."Tank CIP" AND #"CIP Req OK" AND #IN_FBAV_CIP_Tank));
   #Out_AV_Outlet := #alwaysOn AND #Actuator.AV_Outlet;
END_REGION

REGION Network 23: AV Transfer
   RUNG wire#powerrail
      Contact( #alwaysOn )
      wire#w1
      Contact( #state."Ready for Transfer" )
      Contact( #IN_FBAV_Outlet )
      I_Contact( #AlarmProd_pasteur )
      Coil( #Actuator.AV_Transfer )
   END_RUNG
   RUNG wire#w1
      Contact( #Actuator.AV_Transfer )
      Coil( #Out_AV_Transfer )
   END_RUNG
   // the same network as SCL:
   #Actuator.AV_Transfer := #alwaysOn AND #state."Ready for Transfer" AND #IN_FBAV_Outlet AND NOT #AlarmProd_pasteur;
   #Out_AV_Transfer := #alwaysOn AND #Actuator.AV_Transfer;
END_REGION

REGION Network 24: AV CIP Tank
   RUNG wire#powerrail
      Contact( #alwaysOn )
      wire#w1
      Contact( #state."Tank CIP" )
      Contact( #"CIP Req OK" )
      Coil( #Actuator.AV_CIP_Tank )
   END_RUNG
   RUNG wire#w1
      Contact( #Actuator.AV_CIP_Tank )
      Coil( #Out_AV_CIP_Tank )
   END_RUNG
   // the same network as SCL:
   #Actuator.AV_CIP_Tank := #alwaysOn AND #state."Tank CIP" AND #"CIP Req OK";
   #Out_AV_CIP_Tank := #alwaysOn AND #Actuator.AV_CIP_Tank;
END_REGION

REGION Network 25: AV CIP Line
   RUNG wire#powerrail
      Contact( #alwaysOn )
      wire#w1
      Contact( #state."Line CIP" )
      Contact( #"CIP Req OK" )
      Coil( #Actuator.AV_CIP_Line )
   END_RUNG
   RUNG wire#w1
      Contact( #Actuator.AV_CIP_Line )
      Coil( #Out_AV_CIP_Line )
   END_RUNG
   // the same network as SCL:
   #Actuator.AV_CIP_Line := #alwaysOn AND #state."Line CIP" AND #"CIP Req OK";
   #Out_AV_CIP_Line := #alwaysOn AND #Actuator.AV_CIP_Line;
END_REGION

REGION Network 27: Pump Transfer
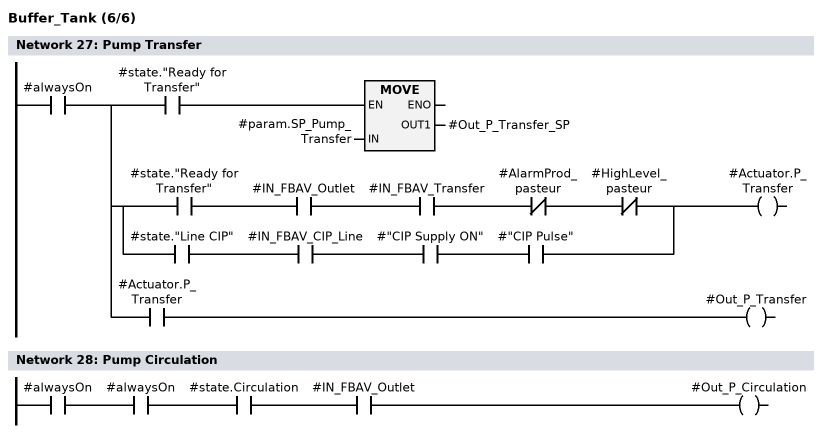
   RUNG wire#powerrail
      Contact( #alwaysOn )
      wire#w1
      Contact( #state."Ready for Transfer" )
      Move(in := #param.SP_Pump_Transfer, out1 => #Out_P_Transfer_SP)
   END_RUNG
   RUNG wire#w1
      Contact( #state."Ready for Transfer" )
      Contact( #IN_FBAV_Outlet )
      Contact( #IN_FBAV_Transfer )
      I_Contact( #AlarmProd_pasteur )
      I_Contact( #HighLevel_pasteur )
      wire#w2
      Coil( #Actuator.P_Transfer )
   END_RUNG
   RUNG wire#w1
      Contact( #state."Line CIP" )
      Contact( #IN_FBAV_CIP_Line )
      Contact( #"CIP Supply ON" )
      Contact( #"CIP Pulse" )
   END_RUNG wire#w2
   RUNG wire#w1
      Contact( #Actuator.P_Transfer )
      Coil( #Out_P_Transfer )
   END_RUNG
   // the same network as SCL:
   IF #alwaysOn AND #state."Ready for Transfer" THEN #Out_P_Transfer_SP := #param.SP_Pump_Transfer; END_IF;
   #Actuator.P_Transfer := #alwaysOn AND ((#state."Ready for Transfer" AND #IN_FBAV_Outlet AND #IN_FBAV_Transfer AND NOT #AlarmProd_pasteur AND NOT #HighLevel_pasteur) OR (#state."Line CIP" AND #IN_FBAV_CIP_Line AND #"CIP Supply ON" AND #"CIP Pulse"));
   #Out_P_Transfer := #alwaysOn AND #Actuator.P_Transfer;
END_REGION

REGION Network 28: Pump Circulation
   RUNG wire#powerrail
      Contact( #alwaysOn )
      Contact( #alwaysOn )
      Contact( #state.Circulation )
      Contact( #IN_FBAV_Outlet )
      Coil( #Out_P_Circulation )
   END_RUNG
   // the same network as SCL:
   #Out_P_Circulation := #alwaysOn AND #alwaysOn AND #state.Circulation AND #IN_FBAV_Outlet;
END_REGION
END_FUNCTION_BLOCK

FUNCTION_BLOCK "IO_Valve_Buffer"   // FB19, LAD
{ S7_Optimized_Access := 'FALSE' }
VERSION : 0.1
// stored: AutoNumber true, IsIECCheckEnabled false, SetENOAutomatically false, UDAEnableTagReadback false
   VAR_INPUT
      "lock 1" : Bool;
      "lock 2" : Bool;
      "lock 3" : Bool;
      "lock 4" : Bool;
      init : Bool;
      reset : Bool;
      testing : Bool;
   END_VAR
   VAR
      "AV-22.11" : "Valve";
      "AV-22.21" : "Valve";
      "AV-22.22" : "Valve";
      "AV-22.23" : "Valve";
      "AV-32.01" : "Valve";
      "AV-32.02" : "Valve";
      "AV-32.03" : "Valve";
      "AV-32.04" : "Valve";
      "AV-32.11" : "Valve";
      "AV-32.21" : "Valve";
      "AV-32.22" : "Valve";
      "AV-32.23" : "Valve";
      "AV-61.01" : "Valve";
      "AV-61.02" : "Valve";
      "AV-61.03" : "Valve";
      "AV-61.04" : "Valve";
      "AV-61.05" : "Valve";
      "AV-61.21" : "Valve";
      "AV-62.06" : "Valve";
      "AV-64.01" : "Valve";
      "AV-64.02" : "Valve";
      "AV-64.03" : "Valve";
      "AV-64.04" : "Valve";
      "AV-64.05" : "Valve";
      "AV-64.06" : "Valve";
      "AV-65.01" : "Valve";
      "AV-65.02" : "Valve";
      "AV-65.03" : "Valve";
      "AV-65.04" : "Valve";
      "AV-65.05" : "Valve";
      "AV-65.21" : "Valve";
      "AV-66.01" : "Valve";
      "AV-66.02" : "Valve";
      "AV-66.03" : "Valve";
      "AV-66.04" : "Valve";
      "AV-66.05" : "Valve";
      "AV-66.06" : "Valve";
      "AV-67.01" : "Valve";
      "AV-67.02" : "Valve";
      "AV-67.03" : "Valve";
      "AV-67.04" : "Valve";
      "AV-67.05" : "Valve";
      "AV-68.01" : "Valve";
      "AV-68.02" : "Valve";
      "AV-68.03" : "Valve";
      "AV-68.04" : "Valve";
      "AV-68.05" : "Valve";
      "AV-68.06" : "Valve";
   END_VAR
BEGIN

REGION Network 1 (SCL): FB OPEN AND CLOSE VALVE T-22
   IF #testing THEN
       // Statement section IF
       #"AV-22.11".FB_OPEN := #"AV-22.11".QCMD_OP;
       #"AV-22.11".FB_CLOSE := NOT #"AV-22.11".QCMD_OP;
       #"AV-22.21".FB_OPEN := #"AV-22.21".QCMD_OP;
       #"AV-22.21".FB_CLOSE := NOT #"AV-22.21".QCMD_OP;
       #"AV-22.22".FB_OPEN := #"AV-22.22".QCMD_OP;
       #"AV-22.22".FB_CLOSE := NOT #"AV-22.22".QCMD_OP;
       #"AV-22.23".FB_OPEN := #"AV-22.23".QCMD_OP;
       #"AV-22.23".FB_CLOSE := NOT #"AV-22.23".QCMD_OP;
   ELSE
       // Statement section ELSE
       #"AV-22.11".FB_OPEN := #"AV-22.11".QCMD_OP;
       #"AV-22.11".FB_CLOSE := NOT #"AV-22.11".QCMD_OP;
       #"AV-22.21".FB_OPEN := #"AV-22.21".QCMD_OP;
       #"AV-22.21".FB_CLOSE := NOT #"AV-22.21".QCMD_OP;
       #"AV-22.22".FB_OPEN := #"AV-22.22".QCMD_OP;
       #"AV-22.22".FB_CLOSE := NOT #"AV-22.22".QCMD_OP;
       #"AV-22.23".FB_OPEN := #"AV-22.23".QCMD_OP;
       #"AV-22.23".FB_CLOSE := NOT #"AV-22.23".QCMD_OP;
   END_IF;
END_REGION

NETWORK
TITLE = FB MONITORING TIME VALVE T-22
// FB OPEN TIME
      L     T#20s;
      T     #"AV-22.11".MON_T;
      T     #"AV-22.21".MON_T;
      T     #"AV-22.22".MON_T;
      T     #"AV-22.23".MON_T;
// FB CLOSE TIME
      L     T#20s;
      T     #"AV-22.11".MON_T_CLOSE;
      T     #"AV-22.21".MON_T_CLOSE;
      T     #"AV-22.22".MON_T_CLOSE;
      T     #"AV-22.23".MON_T_CLOSE;


REGION Network 3: AV-22.11
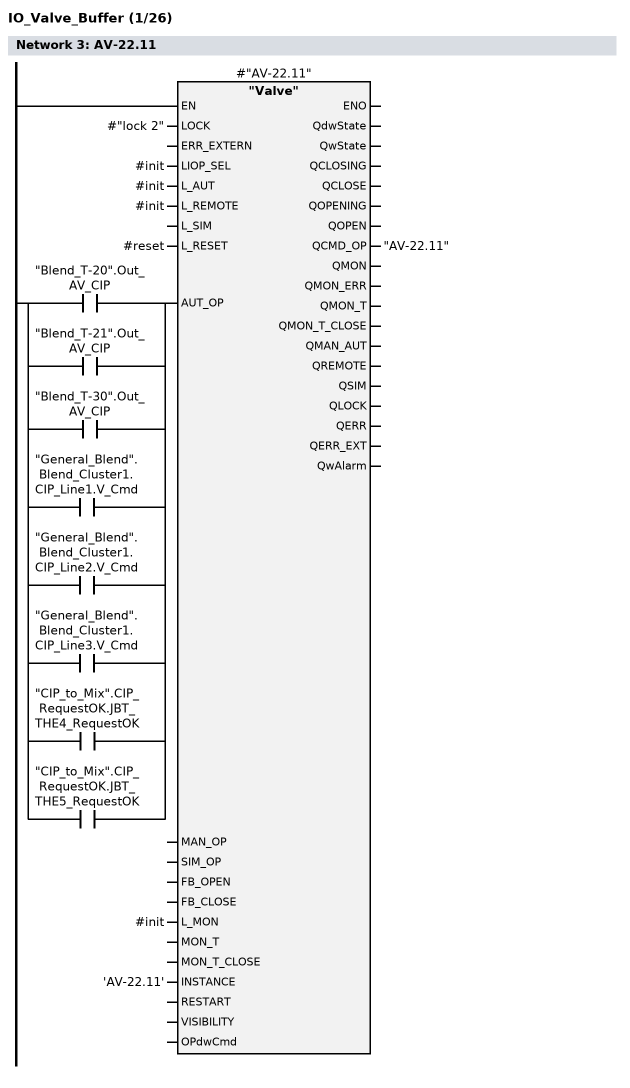
   RUNG wire#powerrail
      #"AV-22.11"(AUT_OP := wire#w1, LOCK := #"lock 2", ERR_EXTERN :=, LIOP_SEL := #init, L_AUT := #init, L_REMOTE := #init, L_SIM :=, L_RESET := #reset, MAN_OP :=, SIM_OP :=, FB_OPEN :=, FB_CLOSE :=, L_MON := #init, MON_T :=, MON_T_CLOSE :=, INSTANCE := 'AV-22.11', RESTART :=, VISIBILITY :=, OPdwCmd :=, QdwState =>, QwState =>, QCLOSING =>, QCLOSE =>, QOPENING =>, QOPEN =>, QCMD_OP => "AV-22.11", QMON =>, QMON_ERR =>, QMON_T =>, QMON_T_CLOSE =>, QMAN_AUT =>, QREMOTE =>, QSIM =>, QLOCK =>, QERR =>, QERR_EXT =>, QwAlarm =>)
   END_RUNG
   RUNG wire#powerrail
      Contact( "Blend_T-20".Out_AV_CIP )
   END_RUNG wire#w1
   RUNG wire#powerrail
      Contact( "Blend_T-21".Out_AV_CIP )
   END_RUNG wire#w1
   RUNG wire#powerrail
      Contact( "Blend_T-30".Out_AV_CIP )
   END_RUNG wire#w1
   RUNG wire#powerrail
      Contact( "General_Blend".Blend_Cluster1.CIP_Line1.V_Cmd )
   END_RUNG wire#w1
   RUNG wire#powerrail
      Contact( "General_Blend".Blend_Cluster1.CIP_Line2.V_Cmd )
   END_RUNG wire#w1
   RUNG wire#powerrail
      Contact( "General_Blend".Blend_Cluster1.CIP_Line3.V_Cmd )
   END_RUNG wire#w1
   RUNG wire#powerrail
      Contact( "CIP_to_Mix".CIP_RequestOK.JBT_THE4_RequestOK )
   END_RUNG wire#w1
   RUNG wire#powerrail
      Contact( "CIP_to_Mix".CIP_RequestOK.JBT_THE5_RequestOK )
   END_RUNG wire#w1
   // the same network as SCL:
   #"AV-22.11"(LOCK := #"lock 2",   // "Valve"
               LIOP_SEL := #init,
               L_AUT := #init,
               L_REMOTE := #init,
               L_RESET := #reset,
               AUT_OP := "Blend_T-20".Out_AV_CIP OR "Blend_T-21".Out_AV_CIP OR "Blend_T-30".Out_AV_CIP OR "General_Blend".Blend_Cluster1.CIP_Line1.V_Cmd OR "General_Blend".Blend_Cluster1.CIP_Line2.V_Cmd OR "General_Blend".Blend_Cluster1.CIP_Line3.V_Cmd OR "CIP_to_Mix".CIP_RequestOK.JBT_THE4_RequestOK OR "CIP_to_Mix".CIP_RequestOK.JBT_THE5_RequestOK,
               L_MON := #init,
               INSTANCE := 'AV-22.11',
               QCMD_OP => "AV-22.11");
END_REGION

REGION Network 4: AV-22.21
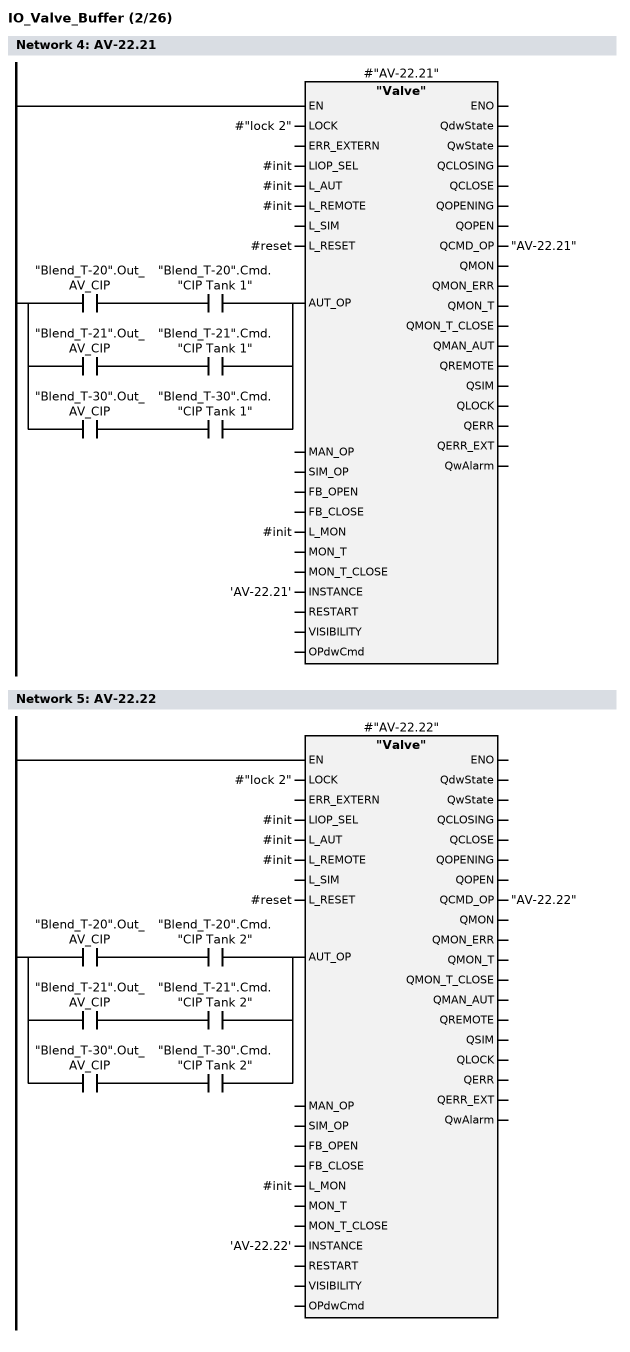
   RUNG wire#powerrail
      #"AV-22.21"(AUT_OP := wire#w1, LOCK := #"lock 2", ERR_EXTERN :=, LIOP_SEL := #init, L_AUT := #init, L_REMOTE := #init, L_SIM :=, L_RESET := #reset, MAN_OP :=, SIM_OP :=, FB_OPEN :=, FB_CLOSE :=, L_MON := #init, MON_T :=, MON_T_CLOSE :=, INSTANCE := 'AV-22.21', RESTART :=, VISIBILITY :=, OPdwCmd :=, QdwState =>, QwState =>, QCLOSING =>, QCLOSE =>, QOPENING =>, QOPEN =>, QCMD_OP => "AV-22.21", QMON =>, QMON_ERR =>, QMON_T =>, QMON_T_CLOSE =>, QMAN_AUT =>, QREMOTE =>, QSIM =>, QLOCK =>, QERR =>, QERR_EXT =>, QwAlarm =>)
   END_RUNG
   RUNG wire#powerrail
      Contact( "Blend_T-20".Out_AV_CIP )
      Contact( "Blend_T-20".Cmd."CIP Tank 1" )
   END_RUNG wire#w1
   RUNG wire#powerrail
      Contact( "Blend_T-21".Out_AV_CIP )
      Contact( "Blend_T-21".Cmd."CIP Tank 1" )
   END_RUNG wire#w1
   RUNG wire#powerrail
      Contact( "Blend_T-30".Out_AV_CIP )
      Contact( "Blend_T-30".Cmd."CIP Tank 1" )
   END_RUNG wire#w1
   // the same network as SCL:
   #"AV-22.21"(LOCK := #"lock 2",   // "Valve"
               LIOP_SEL := #init,
               L_AUT := #init,
               L_REMOTE := #init,
               L_RESET := #reset,
               AUT_OP := ("Blend_T-20".Out_AV_CIP AND "Blend_T-20".Cmd."CIP Tank 1") OR ("Blend_T-21".Out_AV_CIP AND "Blend_T-21".Cmd."CIP Tank 1") OR ("Blend_T-30".Out_AV_CIP AND "Blend_T-30".Cmd."CIP Tank 1"),
               L_MON := #init,
               INSTANCE := 'AV-22.21',
               QCMD_OP => "AV-22.21");
END_REGION

REGION Network 5: AV-22.22
   RUNG wire#powerrail
      #"AV-22.22"(AUT_OP := wire#w1, LOCK := #"lock 2", ERR_EXTERN :=, LIOP_SEL := #init, L_AUT := #init, L_REMOTE := #init, L_SIM :=, L_RESET := #reset, MAN_OP :=, SIM_OP :=, FB_OPEN :=, FB_CLOSE :=, L_MON := #init, MON_T :=, MON_T_CLOSE :=, INSTANCE := 'AV-22.22', RESTART :=, VISIBILITY :=, OPdwCmd :=, QdwState =>, QwState =>, QCLOSING =>, QCLOSE =>, QOPENING =>, QOPEN =>, QCMD_OP => "AV-22.22", QMON =>, QMON_ERR =>, QMON_T =>, QMON_T_CLOSE =>, QMAN_AUT =>, QREMOTE =>, QSIM =>, QLOCK =>, QERR =>, QERR_EXT =>, QwAlarm =>)
   END_RUNG
   RUNG wire#powerrail
      Contact( "Blend_T-20".Out_AV_CIP )
      Contact( "Blend_T-20".Cmd."CIP Tank 2" )
   END_RUNG wire#w1
   RUNG wire#powerrail
      Contact( "Blend_T-21".Out_AV_CIP )
      Contact( "Blend_T-21".Cmd."CIP Tank 2" )
   END_RUNG wire#w1
   RUNG wire#powerrail
      Contact( "Blend_T-30".Out_AV_CIP )
      Contact( "Blend_T-30".Cmd."CIP Tank 2" )
   END_RUNG wire#w1
   // the same network as SCL:
   #"AV-22.22"(LOCK := #"lock 2",   // "Valve"
               LIOP_SEL := #init,
               L_AUT := #init,
               L_REMOTE := #init,
               L_RESET := #reset,
               AUT_OP := ("Blend_T-20".Out_AV_CIP AND "Blend_T-20".Cmd."CIP Tank 2") OR ("Blend_T-21".Out_AV_CIP AND "Blend_T-21".Cmd."CIP Tank 2") OR ("Blend_T-30".Out_AV_CIP AND "Blend_T-30".Cmd."CIP Tank 2"),
               L_MON := #init,
               INSTANCE := 'AV-22.22',
               QCMD_OP => "AV-22.22");
END_REGION

REGION Network 6: AV-22.23
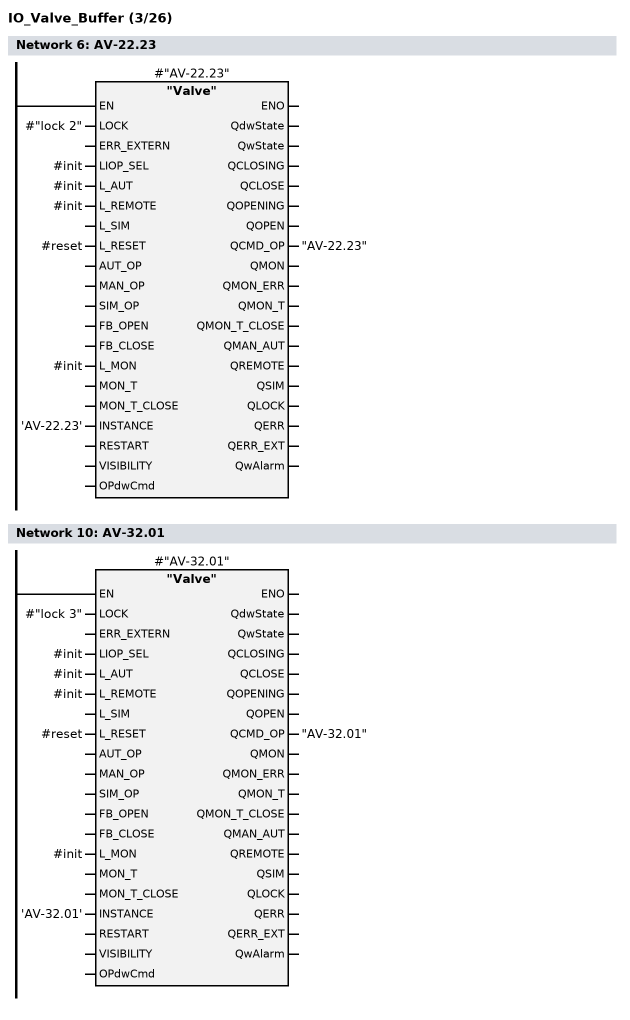
   RUNG wire#powerrail
      #"AV-22.23"(LOCK := #"lock 2", ERR_EXTERN :=, LIOP_SEL := #init, L_AUT := #init, L_REMOTE := #init, L_SIM :=, L_RESET := #reset, AUT_OP :=, MAN_OP :=, SIM_OP :=, FB_OPEN :=, FB_CLOSE :=, L_MON := #init, MON_T :=, MON_T_CLOSE :=, INSTANCE := 'AV-22.23', RESTART :=, VISIBILITY :=, OPdwCmd :=, QdwState =>, QwState =>, QCLOSING =>, QCLOSE =>, QOPENING =>, QOPEN =>, QCMD_OP => "AV-22.23", QMON =>, QMON_ERR =>, QMON_T =>, QMON_T_CLOSE =>, QMAN_AUT =>, QREMOTE =>, QSIM =>, QLOCK =>, QERR =>, QERR_EXT =>, QwAlarm =>)
   END_RUNG
   // the same network as SCL:
   #"AV-22.23"(LOCK := #"lock 2",   // "Valve"
               LIOP_SEL := #init,
               L_AUT := #init,
               L_REMOTE := #init,
               L_RESET := #reset,
               L_MON := #init,
               INSTANCE := 'AV-22.23',
               QCMD_OP => "AV-22.23");
END_REGION

REGION Network 8 (SCL): FB OPEN AND CLOSE VALVE T-32
   IF #testing THEN
       // Statement section IF
       #"AV-32.01".FB_OPEN := #"AV-32.01".QCMD_OP;
       #"AV-32.01".FB_CLOSE := NOT #"AV-32.01".QCMD_OP;
       #"AV-32.02".FB_OPEN := #"AV-32.02".QCMD_OP;
       #"AV-32.02".FB_CLOSE := NOT #"AV-32.02".QCMD_OP;
       #"AV-32.03".FB_OPEN := #"AV-32.03".QCMD_OP;
       #"AV-32.03".FB_CLOSE := NOT #"AV-32.03".QCMD_OP;
       #"AV-32.04".FB_OPEN := #"AV-32.04".QCMD_OP;
       #"AV-32.04".FB_CLOSE := NOT #"AV-32.04".QCMD_OP;
       #"AV-32.11".FB_OPEN := #"AV-32.11".QCMD_OP;
       #"AV-32.11".FB_CLOSE := NOT #"AV-32.11".QCMD_OP;
       #"AV-32.21".FB_OPEN := #"AV-32.21".QCMD_OP;
       #"AV-32.21".FB_CLOSE := NOT #"AV-32.21".QCMD_OP;
       #"AV-32.22".FB_OPEN := #"AV-32.22".QCMD_OP;
       #"AV-32.22".FB_CLOSE := NOT #"AV-32.22".QCMD_OP;
       #"AV-32.23".FB_OPEN := #"AV-32.23".QCMD_OP;
       #"AV-32.23".FB_CLOSE := NOT #"AV-32.23".QCMD_OP;
   ELSE
       // Statement section ELSE
       #"AV-32.01".FB_OPEN := #"AV-32.01".QCMD_OP;
       #"AV-32.01".FB_CLOSE := NOT #"AV-32.01".QCMD_OP;
       #"AV-32.02".FB_OPEN := #"AV-32.02".QCMD_OP;
       #"AV-32.02".FB_CLOSE := NOT #"AV-32.02".QCMD_OP;
       #"AV-32.03".FB_OPEN := #"AV-32.03".QCMD_OP;
       #"AV-32.03".FB_CLOSE := NOT #"AV-32.03".QCMD_OP;
       #"AV-32.04".FB_OPEN := #"AV-32.04".QCMD_OP;
       #"AV-32.04".FB_CLOSE := NOT #"AV-32.04".QCMD_OP;
       #"AV-32.11".FB_OPEN := #"AV-32.11".QCMD_OP;
       #"AV-32.11".FB_CLOSE := NOT #"AV-32.11".QCMD_OP;
       #"AV-32.21".FB_OPEN := #"AV-32.21".QCMD_OP;
       #"AV-32.21".FB_CLOSE := NOT #"AV-32.21".QCMD_OP;
       #"AV-32.22".FB_OPEN := #"AV-32.22".QCMD_OP;
       #"AV-32.22".FB_CLOSE := NOT #"AV-32.22".QCMD_OP;
       #"AV-32.23".FB_OPEN := #"AV-32.23".QCMD_OP;
       #"AV-32.23".FB_CLOSE := NOT #"AV-32.23".QCMD_OP;
   END_IF;
END_REGION

NETWORK
TITLE = FB MONITORING TIME VALVE T-32
// FB OPEN TIME
      L     T#20s;
      T     #"AV-32.01".MON_T;
      T     #"AV-32.02".MON_T;
      T     #"AV-32.03".MON_T;
      T     #"AV-32.04".MON_T;
      T     #"AV-32.11".MON_T;
      T     #"AV-32.21".MON_T;
      T     #"AV-32.22".MON_T;
      T     #"AV-32.23".MON_T;
// FB CLOSE TIME
      L     T#20s;
      T     #"AV-32.01".MON_T_CLOSE;
      T     #"AV-32.02".MON_T_CLOSE;
      T     #"AV-32.03".MON_T_CLOSE;
      T     #"AV-32.04".MON_T_CLOSE;
      T     #"AV-32.11".MON_T_CLOSE;
      T     #"AV-32.21".MON_T_CLOSE;
      T     #"AV-32.22".MON_T_CLOSE;
      T     #"AV-32.23".MON_T_CLOSE;


REGION Network 10: AV-32.01
   RUNG wire#powerrail
      #"AV-32.01"(LOCK := #"lock 3", ERR_EXTERN :=, LIOP_SEL := #init, L_AUT := #init, L_REMOTE := #init, L_SIM :=, L_RESET := #reset, AUT_OP :=, MAN_OP :=, SIM_OP :=, FB_OPEN :=, FB_CLOSE :=, L_MON := #init, MON_T :=, MON_T_CLOSE :=, INSTANCE := 'AV-32.01', RESTART :=, VISIBILITY :=, OPdwCmd :=, QdwState =>, QwState =>, QCLOSING =>, QCLOSE =>, QOPENING =>, QOPEN =>, QCMD_OP => "AV-32.01", QMON =>, QMON_ERR =>, QMON_T =>, QMON_T_CLOSE =>, QMAN_AUT =>, QREMOTE =>, QSIM =>, QLOCK =>, QERR =>, QERR_EXT =>, QwAlarm =>)
   END_RUNG
   // the same network as SCL:
   #"AV-32.01"(LOCK := #"lock 3",   // "Valve"
               LIOP_SEL := #init,
               L_AUT := #init,
               L_REMOTE := #init,
               L_RESET := #reset,
               L_MON := #init,
               INSTANCE := 'AV-32.01',
               QCMD_OP => "AV-32.01");
END_REGION

REGION Network 11: AV-32.02
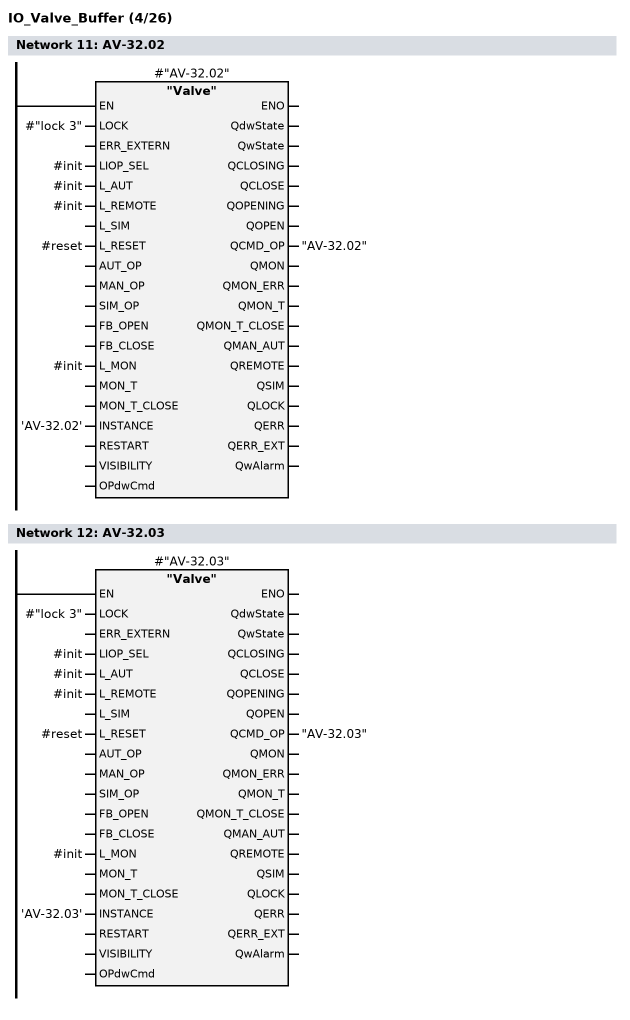
   RUNG wire#powerrail
      #"AV-32.02"(LOCK := #"lock 3", ERR_EXTERN :=, LIOP_SEL := #init, L_AUT := #init, L_REMOTE := #init, L_SIM :=, L_RESET := #reset, AUT_OP :=, MAN_OP :=, SIM_OP :=, FB_OPEN :=, FB_CLOSE :=, L_MON := #init, MON_T :=, MON_T_CLOSE :=, INSTANCE := 'AV-32.02', RESTART :=, VISIBILITY :=, OPdwCmd :=, QdwState =>, QwState =>, QCLOSING =>, QCLOSE =>, QOPENING =>, QOPEN =>, QCMD_OP => "AV-32.02", QMON =>, QMON_ERR =>, QMON_T =>, QMON_T_CLOSE =>, QMAN_AUT =>, QREMOTE =>, QSIM =>, QLOCK =>, QERR =>, QERR_EXT =>, QwAlarm =>)
   END_RUNG
   // the same network as SCL:
   #"AV-32.02"(LOCK := #"lock 3",   // "Valve"
               LIOP_SEL := #init,
               L_AUT := #init,
               L_REMOTE := #init,
               L_RESET := #reset,
               L_MON := #init,
               INSTANCE := 'AV-32.02',
               QCMD_OP => "AV-32.02");
END_REGION

REGION Network 12: AV-32.03
   RUNG wire#powerrail
      #"AV-32.03"(LOCK := #"lock 3", ERR_EXTERN :=, LIOP_SEL := #init, L_AUT := #init, L_REMOTE := #init, L_SIM :=, L_RESET := #reset, AUT_OP :=, MAN_OP :=, SIM_OP :=, FB_OPEN :=, FB_CLOSE :=, L_MON := #init, MON_T :=, MON_T_CLOSE :=, INSTANCE := 'AV-32.03', RESTART :=, VISIBILITY :=, OPdwCmd :=, QdwState =>, QwState =>, QCLOSING =>, QCLOSE =>, QOPENING =>, QOPEN =>, QCMD_OP => "AV-32.03", QMON =>, QMON_ERR =>, QMON_T =>, QMON_T_CLOSE =>, QMAN_AUT =>, QREMOTE =>, QSIM =>, QLOCK =>, QERR =>, QERR_EXT =>, QwAlarm =>)
   END_RUNG
   // the same network as SCL:
   #"AV-32.03"(LOCK := #"lock 3",   // "Valve"
               LIOP_SEL := #init,
               L_AUT := #init,
               L_REMOTE := #init,
               L_RESET := #reset,
               L_MON := #init,
               INSTANCE := 'AV-32.03',
               QCMD_OP => "AV-32.03");
END_REGION

REGION Network 13: AV-32.04
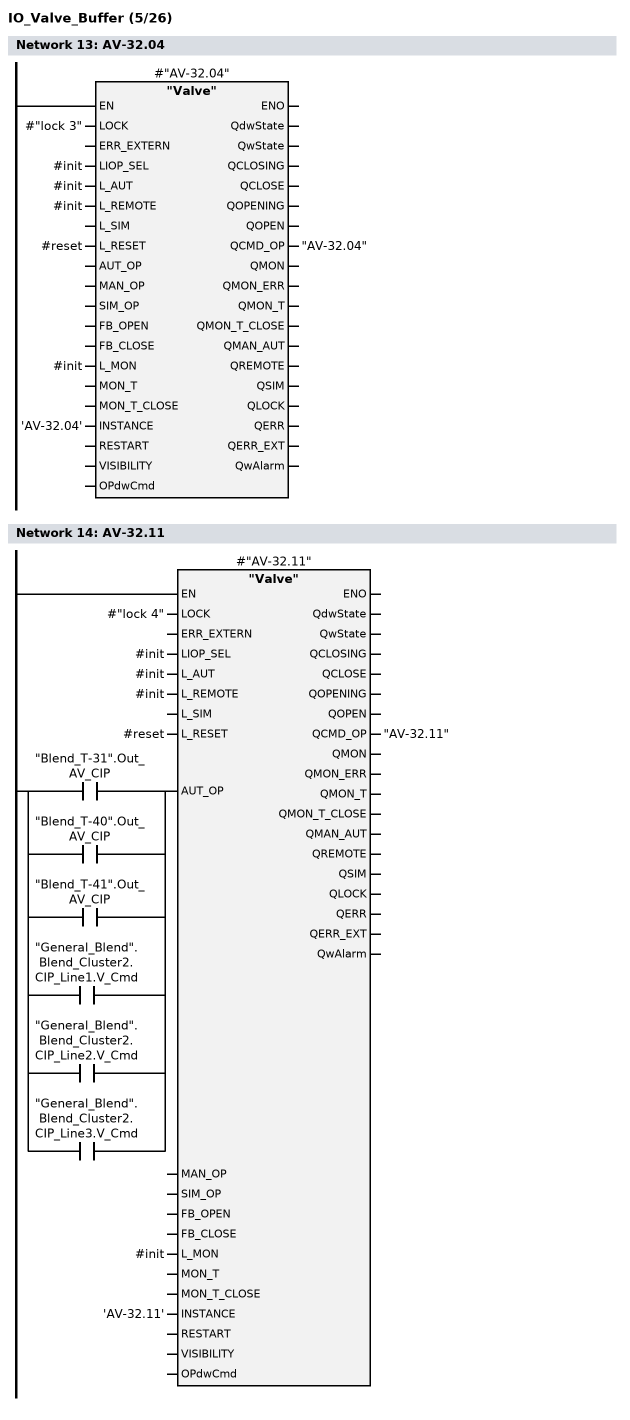
   RUNG wire#powerrail
      #"AV-32.04"(LOCK := #"lock 3", ERR_EXTERN :=, LIOP_SEL := #init, L_AUT := #init, L_REMOTE := #init, L_SIM :=, L_RESET := #reset, AUT_OP :=, MAN_OP :=, SIM_OP :=, FB_OPEN :=, FB_CLOSE :=, L_MON := #init, MON_T :=, MON_T_CLOSE :=, INSTANCE := 'AV-32.04', RESTART :=, VISIBILITY :=, OPdwCmd :=, QdwState =>, QwState =>, QCLOSING =>, QCLOSE =>, QOPENING =>, QOPEN =>, QCMD_OP => "AV-32.04", QMON =>, QMON_ERR =>, QMON_T =>, QMON_T_CLOSE =>, QMAN_AUT =>, QREMOTE =>, QSIM =>, QLOCK =>, QERR =>, QERR_EXT =>, QwAlarm =>)
   END_RUNG
   // the same network as SCL:
   #"AV-32.04"(LOCK := #"lock 3",   // "Valve"
               LIOP_SEL := #init,
               L_AUT := #init,
               L_REMOTE := #init,
               L_RESET := #reset,
               L_MON := #init,
               INSTANCE := 'AV-32.04',
               QCMD_OP => "AV-32.04");
END_REGION

REGION Network 14: AV-32.11
   RUNG wire#powerrail
      #"AV-32.11"(AUT_OP := wire#w1, LOCK := #"lock 4", ERR_EXTERN :=, LIOP_SEL := #init, L_AUT := #init, L_REMOTE := #init, L_SIM :=, L_RESET := #reset, MAN_OP :=, SIM_OP :=, FB_OPEN :=, FB_CLOSE :=, L_MON := #init, MON_T :=, MON_T_CLOSE :=, INSTANCE := 'AV-32.11', RESTART :=, VISIBILITY :=, OPdwCmd :=, QdwState =>, QwState =>, QCLOSING =>, QCLOSE =>, QOPENING =>, QOPEN =>, QCMD_OP => "AV-32.11", QMON =>, QMON_ERR =>, QMON_T =>, QMON_T_CLOSE =>, QMAN_AUT =>, QREMOTE =>, QSIM =>, QLOCK =>, QERR =>, QERR_EXT =>, QwAlarm =>)
   END_RUNG
   RUNG wire#powerrail
      Contact( "Blend_T-31".Out_AV_CIP )
   END_RUNG wire#w1
   RUNG wire#powerrail
      Contact( "Blend_T-40".Out_AV_CIP )
   END_RUNG wire#w1
   RUNG wire#powerrail
      Contact( "Blend_T-41".Out_AV_CIP )
   END_RUNG wire#w1
   RUNG wire#powerrail
      Contact( "General_Blend".Blend_Cluster2.CIP_Line1.V_Cmd )
   END_RUNG wire#w1
   RUNG wire#powerrail
      Contact( "General_Blend".Blend_Cluster2.CIP_Line2.V_Cmd )
   END_RUNG wire#w1
   RUNG wire#powerrail
      Contact( "General_Blend".Blend_Cluster2.CIP_Line3.V_Cmd )
   END_RUNG wire#w1
   // the same network as SCL:
   #"AV-32.11"(LOCK := #"lock 4",   // "Valve"
               LIOP_SEL := #init,
               L_AUT := #init,
               L_REMOTE := #init,
               L_RESET := #reset,
               AUT_OP := "Blend_T-31".Out_AV_CIP OR "Blend_T-40".Out_AV_CIP OR "Blend_T-41".Out_AV_CIP OR "General_Blend".Blend_Cluster2.CIP_Line1.V_Cmd OR "General_Blend".Blend_Cluster2.CIP_Line2.V_Cmd OR "General_Blend".Blend_Cluster2.CIP_Line3.V_Cmd,
               L_MON := #init,
               INSTANCE := 'AV-32.11',
               QCMD_OP => "AV-32.11");
END_REGION

REGION Network 15: AV-32.21
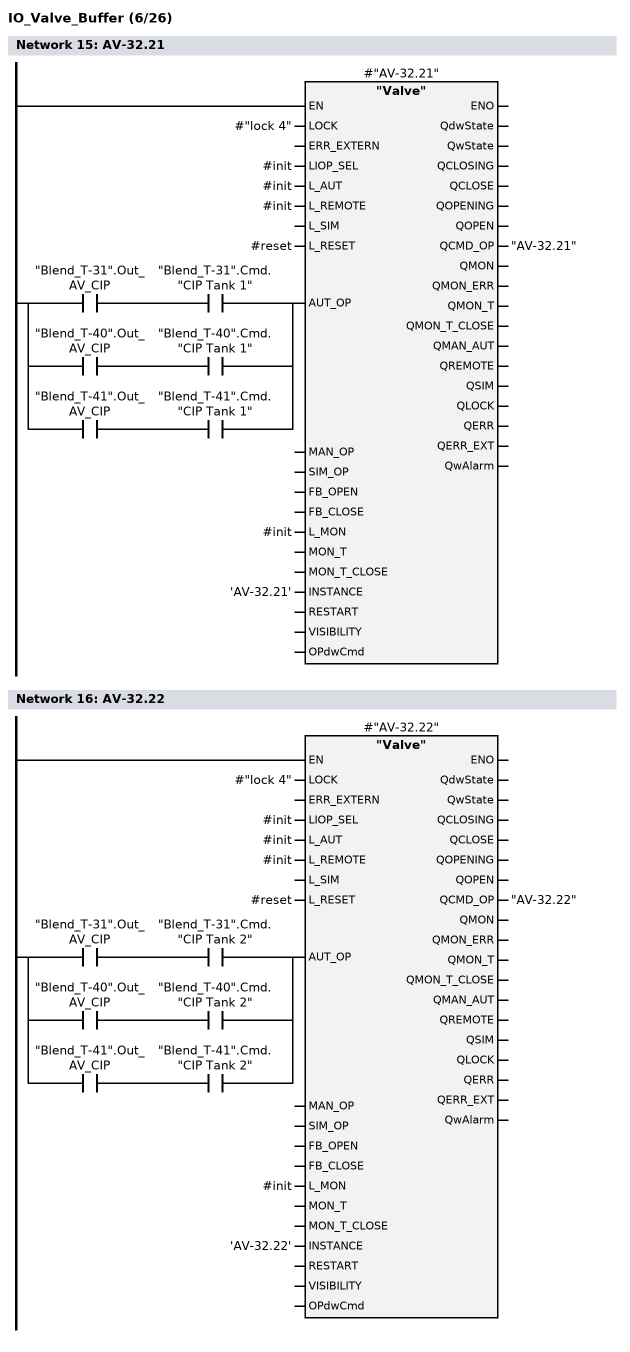
   RUNG wire#powerrail
      #"AV-32.21"(AUT_OP := wire#w1, LOCK := #"lock 4", ERR_EXTERN :=, LIOP_SEL := #init, L_AUT := #init, L_REMOTE := #init, L_SIM :=, L_RESET := #reset, MAN_OP :=, SIM_OP :=, FB_OPEN :=, FB_CLOSE :=, L_MON := #init, MON_T :=, MON_T_CLOSE :=, INSTANCE := 'AV-32.21', RESTART :=, VISIBILITY :=, OPdwCmd :=, QdwState =>, QwState =>, QCLOSING =>, QCLOSE =>, QOPENING =>, QOPEN =>, QCMD_OP => "AV-32.21", QMON =>, QMON_ERR =>, QMON_T =>, QMON_T_CLOSE =>, QMAN_AUT =>, QREMOTE =>, QSIM =>, QLOCK =>, QERR =>, QERR_EXT =>, QwAlarm =>)
   END_RUNG
   RUNG wire#powerrail
      Contact( "Blend_T-31".Out_AV_CIP )
      Contact( "Blend_T-31".Cmd."CIP Tank 1" )
   END_RUNG wire#w1
   RUNG wire#powerrail
      Contact( "Blend_T-40".Out_AV_CIP )
      Contact( "Blend_T-40".Cmd."CIP Tank 1" )
   END_RUNG wire#w1
   RUNG wire#powerrail
      Contact( "Blend_T-41".Out_AV_CIP )
      Contact( "Blend_T-41".Cmd."CIP Tank 1" )
   END_RUNG wire#w1
   // the same network as SCL:
   #"AV-32.21"(LOCK := #"lock 4",   // "Valve"
               LIOP_SEL := #init,
               L_AUT := #init,
               L_REMOTE := #init,
               L_RESET := #reset,
               AUT_OP := ("Blend_T-31".Out_AV_CIP AND "Blend_T-31".Cmd."CIP Tank 1") OR ("Blend_T-40".Out_AV_CIP AND "Blend_T-40".Cmd."CIP Tank 1") OR ("Blend_T-41".Out_AV_CIP AND "Blend_T-41".Cmd."CIP Tank 1"),
               L_MON := #init,
               INSTANCE := 'AV-32.21',
               QCMD_OP => "AV-32.21");
END_REGION

REGION Network 16: AV-32.22
   RUNG wire#powerrail
      #"AV-32.22"(AUT_OP := wire#w1, LOCK := #"lock 4", ERR_EXTERN :=, LIOP_SEL := #init, L_AUT := #init, L_REMOTE := #init, L_SIM :=, L_RESET := #reset, MAN_OP :=, SIM_OP :=, FB_OPEN :=, FB_CLOSE :=, L_MON := #init, MON_T :=, MON_T_CLOSE :=, INSTANCE := 'AV-32.22', RESTART :=, VISIBILITY :=, OPdwCmd :=, QdwState =>, QwState =>, QCLOSING =>, QCLOSE =>, QOPENING =>, QOPEN =>, QCMD_OP => "AV-32.22", QMON =>, QMON_ERR =>, QMON_T =>, QMON_T_CLOSE =>, QMAN_AUT =>, QREMOTE =>, QSIM =>, QLOCK =>, QERR =>, QERR_EXT =>, QwAlarm =>)
   END_RUNG
   RUNG wire#powerrail
      Contact( "Blend_T-31".Out_AV_CIP )
      Contact( "Blend_T-31".Cmd."CIP Tank 2" )
   END_RUNG wire#w1
   RUNG wire#powerrail
      Contact( "Blend_T-40".Out_AV_CIP )
      Contact( "Blend_T-40".Cmd."CIP Tank 2" )
   END_RUNG wire#w1
   RUNG wire#powerrail
      Contact( "Blend_T-41".Out_AV_CIP )
      Contact( "Blend_T-41".Cmd."CIP Tank 2" )
   END_RUNG wire#w1
   // the same network as SCL:
   #"AV-32.22"(LOCK := #"lock 4",   // "Valve"
               LIOP_SEL := #init,
               L_AUT := #init,
               L_REMOTE := #init,
               L_RESET := #reset,
               AUT_OP := ("Blend_T-31".Out_AV_CIP AND "Blend_T-31".Cmd."CIP Tank 2") OR ("Blend_T-40".Out_AV_CIP AND "Blend_T-40".Cmd."CIP Tank 2") OR ("Blend_T-41".Out_AV_CIP AND "Blend_T-41".Cmd."CIP Tank 2"),
               L_MON := #init,
               INSTANCE := 'AV-32.22',
               QCMD_OP => "AV-32.22");
END_REGION

REGION Network 17: AV-32.23
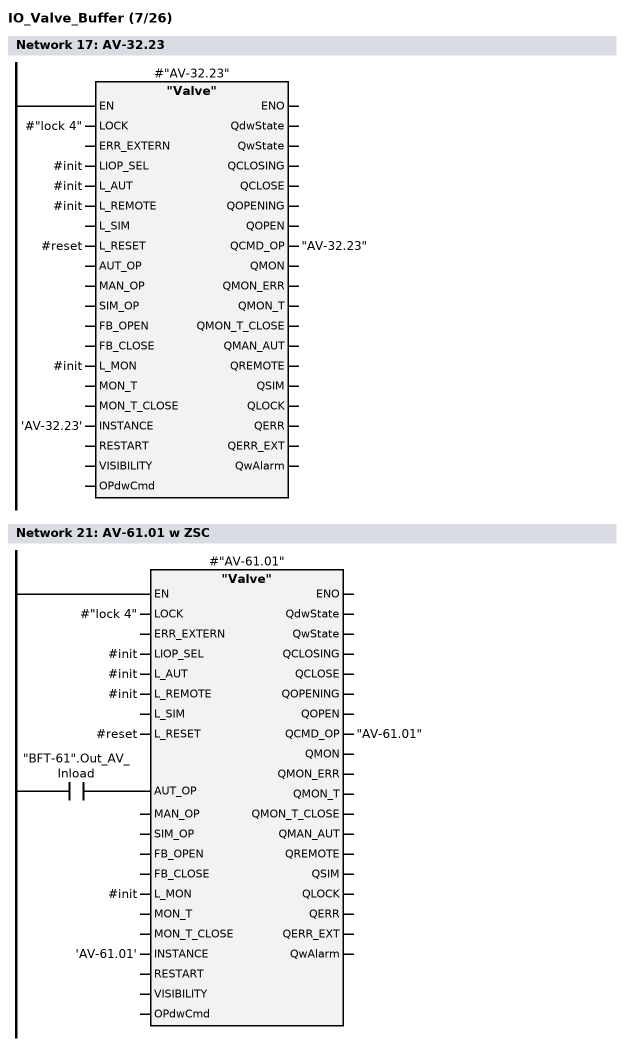
   RUNG wire#powerrail
      #"AV-32.23"(LOCK := #"lock 4", ERR_EXTERN :=, LIOP_SEL := #init, L_AUT := #init, L_REMOTE := #init, L_SIM :=, L_RESET := #reset, AUT_OP :=, MAN_OP :=, SIM_OP :=, FB_OPEN :=, FB_CLOSE :=, L_MON := #init, MON_T :=, MON_T_CLOSE :=, INSTANCE := 'AV-32.23', RESTART :=, VISIBILITY :=, OPdwCmd :=, QdwState =>, QwState =>, QCLOSING =>, QCLOSE =>, QOPENING =>, QOPEN =>, QCMD_OP => "AV-32.23", QMON =>, QMON_ERR =>, QMON_T =>, QMON_T_CLOSE =>, QMAN_AUT =>, QREMOTE =>, QSIM =>, QLOCK =>, QERR =>, QERR_EXT =>, QwAlarm =>)
   END_RUNG
   // the same network as SCL:
   #"AV-32.23"(LOCK := #"lock 4",   // "Valve"
               LIOP_SEL := #init,
               L_AUT := #init,
               L_REMOTE := #init,
               L_RESET := #reset,
               L_MON := #init,
               INSTANCE := 'AV-32.23',
               QCMD_OP => "AV-32.23");
END_REGION

REGION Network 19 (SCL): FB OPEN AND CLOSE VALVE T-61
   IF #testing THEN
       // Statement section IF
       #"AV-61.01".FB_OPEN := #"AV-61.01".QCMD_OP;
       #"AV-61.01".FB_CLOSE := NOT #"AV-61.01".QCMD_OP;
       #"AV-61.02".FB_OPEN := #"AV-61.02".QCMD_OP;
       #"AV-61.02".FB_CLOSE := NOT #"AV-61.02".QCMD_OP;
       #"AV-61.03".FB_OPEN := #"AV-61.03".QCMD_OP;
       #"AV-61.03".FB_CLOSE := NOT #"AV-61.03".QCMD_OP;
       #"AV-61.04".FB_OPEN := #"AV-61.04".QCMD_OP;
       #"AV-61.04".FB_CLOSE := NOT #"AV-61.04".QCMD_OP;
       #"AV-61.05".FB_OPEN := #"AV-61.05".QCMD_OP;
       #"AV-61.05".FB_CLOSE := NOT #"AV-61.05".QCMD_OP;
       #"AV-61.21".FB_OPEN := #"AV-61.21".QCMD_OP;
       #"AV-61.21".FB_CLOSE := NOT #"AV-61.21".QCMD_OP;
   ELSE
       // Statement section ELSE
       #"AV-61.01".FB_OPEN := NOT "ZSC-61.01";
       #"AV-61.01".FB_CLOSE := "ZSC-61.01";
       #"AV-61.02".FB_OPEN := #"AV-61.02".QCMD_OP;
       #"AV-61.02".FB_CLOSE := NOT #"AV-61.02".QCMD_OP;
       #"AV-61.03".FB_OPEN := NOT "ZSC-61.03";
       #"AV-61.03".FB_CLOSE := "ZSC-61.03";
       #"AV-61.04".FB_OPEN := #"AV-61.04".QCMD_OP;
       #"AV-61.04".FB_CLOSE := NOT #"AV-61.04".QCMD_OP;
       #"AV-61.05".FB_OPEN := #"AV-61.05".QCMD_OP;
       #"AV-61.05".FB_CLOSE := NOT #"AV-61.05".QCMD_OP;
       #"AV-61.21".FB_OPEN := #"AV-61.21".QCMD_OP;
       #"AV-61.21".FB_CLOSE := NOT #"AV-61.21".QCMD_OP;
   END_IF;
END_REGION

NETWORK
TITLE = FB MONITORING TIME VALVE T-61
// FB OPEN TIME
      L     T#20s;
      T     #"AV-61.01".MON_T;
      T     #"AV-61.02".MON_T;
      T     #"AV-61.03".MON_T;
      T     #"AV-61.04".MON_T;
      T     #"AV-61.05".MON_T;
      T     #"AV-61.21".MON_T;
// FB CLOSE TIME
      L     T#20s;
      T     #"AV-61.01".MON_T_CLOSE;
      T     #"AV-61.02".MON_T_CLOSE;
      T     #"AV-61.03".MON_T_CLOSE;
      T     #"AV-61.04".MON_T_CLOSE;
      T     #"AV-61.05".MON_T_CLOSE;
      T     #"AV-61.21".MON_T_CLOSE;

REGION Network 21: AV-61.01 w ZSC
   RUNG wire#powerrail
      #"AV-61.01"(AUT_OP := wire#w1, LOCK := #"lock 4", ERR_EXTERN :=, LIOP_SEL := #init, L_AUT := #init, L_REMOTE := #init, L_SIM :=, L_RESET := #reset, MAN_OP :=, SIM_OP :=, FB_OPEN :=, FB_CLOSE :=, L_MON := #init, MON_T :=, MON_T_CLOSE :=, INSTANCE := 'AV-61.01', RESTART :=, VISIBILITY :=, OPdwCmd :=, QdwState =>, QwState =>, QCLOSING =>, QCLOSE =>, QOPENING =>, QOPEN =>, QCMD_OP => "AV-61.01", QMON =>, QMON_ERR =>, QMON_T =>, QMON_T_CLOSE =>, QMAN_AUT =>, QREMOTE =>, QSIM =>, QLOCK =>, QERR =>, QERR_EXT =>, QwAlarm =>)
   END_RUNG
   RUNG wire#powerrail
      Contact( "BFT-61".Out_AV_Inload )
   END_RUNG wire#w1
   // the same network as SCL:
   #"AV-61.01"(LOCK := #"lock 4",   // "Valve"
               LIOP_SEL := #init,
               L_AUT := #init,
               L_REMOTE := #init,
               L_RESET := #reset,
               AUT_OP := "BFT-61".Out_AV_Inload,
               L_MON := #init,
               INSTANCE := 'AV-61.01',
               QCMD_OP => "AV-61.01");
END_REGION

REGION Network 22: AV-61.02
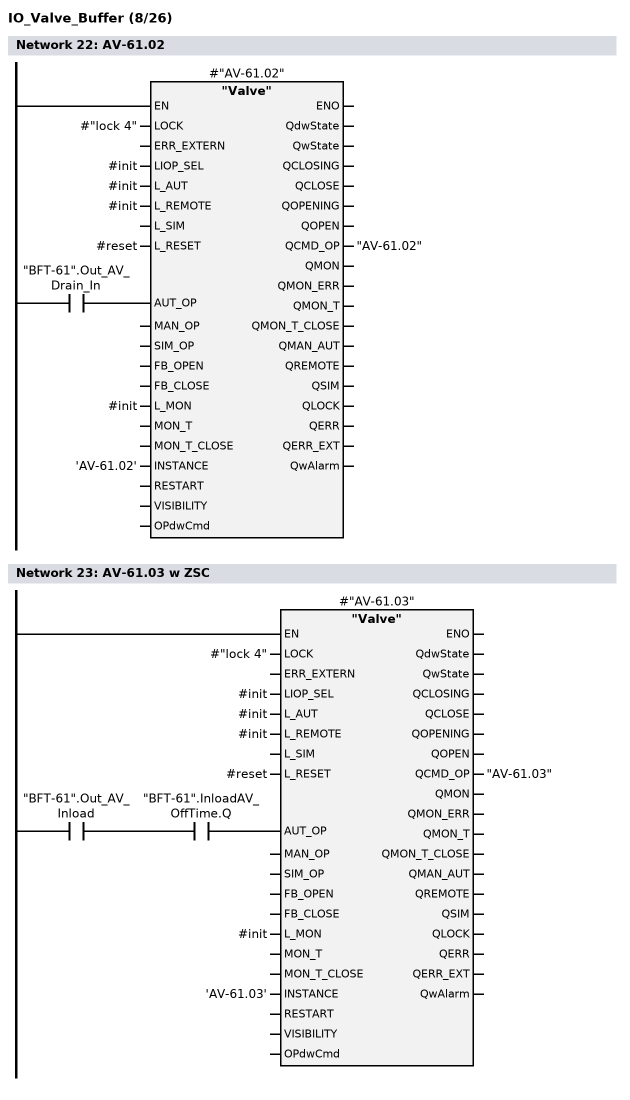
   RUNG wire#powerrail
      #"AV-61.02"(AUT_OP := wire#w1, LOCK := #"lock 4", ERR_EXTERN :=, LIOP_SEL := #init, L_AUT := #init, L_REMOTE := #init, L_SIM :=, L_RESET := #reset, MAN_OP :=, SIM_OP :=, FB_OPEN :=, FB_CLOSE :=, L_MON := #init, MON_T :=, MON_T_CLOSE :=, INSTANCE := 'AV-61.02', RESTART :=, VISIBILITY :=, OPdwCmd :=, QdwState =>, QwState =>, QCLOSING =>, QCLOSE =>, QOPENING =>, QOPEN =>, QCMD_OP => "AV-61.02", QMON =>, QMON_ERR =>, QMON_T =>, QMON_T_CLOSE =>, QMAN_AUT =>, QREMOTE =>, QSIM =>, QLOCK =>, QERR =>, QERR_EXT =>, QwAlarm =>)
   END_RUNG
   RUNG wire#powerrail
      Contact( "BFT-61".Out_AV_Drain_In )
   END_RUNG wire#w1
   // the same network as SCL:
   #"AV-61.02"(LOCK := #"lock 4",   // "Valve"
               LIOP_SEL := #init,
               L_AUT := #init,
               L_REMOTE := #init,
               L_RESET := #reset,
               AUT_OP := "BFT-61".Out_AV_Drain_In,
               L_MON := #init,
               INSTANCE := 'AV-61.02',
               QCMD_OP => "AV-61.02");
END_REGION

REGION Network 23: AV-61.03 w ZSC
   RUNG wire#powerrail
      #"AV-61.03"(AUT_OP := wire#w1, LOCK := #"lock 4", ERR_EXTERN :=, LIOP_SEL := #init, L_AUT := #init, L_REMOTE := #init, L_SIM :=, L_RESET := #reset, MAN_OP :=, SIM_OP :=, FB_OPEN :=, FB_CLOSE :=, L_MON := #init, MON_T :=, MON_T_CLOSE :=, INSTANCE := 'AV-61.03', RESTART :=, VISIBILITY :=, OPdwCmd :=, QdwState =>, QwState =>, QCLOSING =>, QCLOSE =>, QOPENING =>, QOPEN =>, QCMD_OP => "AV-61.03", QMON =>, QMON_ERR =>, QMON_T =>, QMON_T_CLOSE =>, QMAN_AUT =>, QREMOTE =>, QSIM =>, QLOCK =>, QERR =>, QERR_EXT =>, QwAlarm =>)
   END_RUNG
   RUNG wire#powerrail
      Contact( "BFT-61".Out_AV_Inload )
      Contact( "BFT-61".InloadAV_OffTime.Q )
   END_RUNG wire#w1
   // the same network as SCL:
   #"AV-61.03"(LOCK := #"lock 4",   // "Valve"
               LIOP_SEL := #init,
               L_AUT := #init,
               L_REMOTE := #init,
               L_RESET := #reset,
               AUT_OP := "BFT-61".Out_AV_Inload AND "BFT-61".InloadAV_OffTime.Q,
               L_MON := #init,
               INSTANCE := 'AV-61.03',
               QCMD_OP => "AV-61.03");
END_REGION

REGION Network 24: AV-61.04
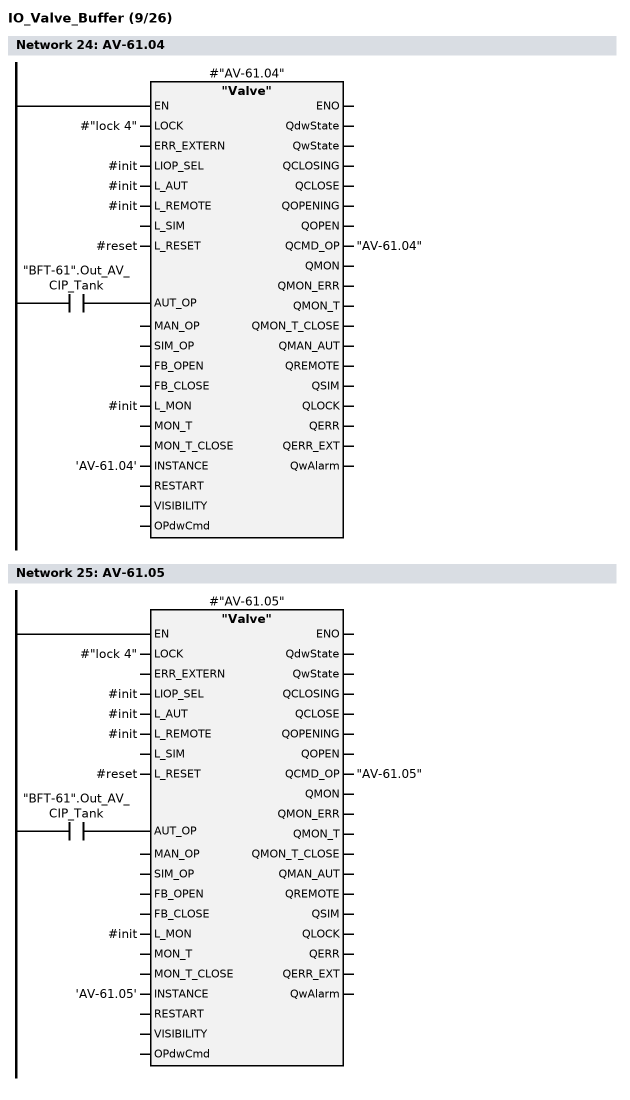
   RUNG wire#powerrail
      #"AV-61.04"(AUT_OP := wire#w1, LOCK := #"lock 4", ERR_EXTERN :=, LIOP_SEL := #init, L_AUT := #init, L_REMOTE := #init, L_SIM :=, L_RESET := #reset, MAN_OP :=, SIM_OP :=, FB_OPEN :=, FB_CLOSE :=, L_MON := #init, MON_T :=, MON_T_CLOSE :=, INSTANCE := 'AV-61.04', RESTART :=, VISIBILITY :=, OPdwCmd :=, QdwState =>, QwState =>, QCLOSING =>, QCLOSE =>, QOPENING =>, QOPEN =>, QCMD_OP => "AV-61.04", QMON =>, QMON_ERR =>, QMON_T =>, QMON_T_CLOSE =>, QMAN_AUT =>, QREMOTE =>, QSIM =>, QLOCK =>, QERR =>, QERR_EXT =>, QwAlarm =>)
   END_RUNG
   RUNG wire#powerrail
      Contact( "BFT-61".Out_AV_CIP_Tank )
   END_RUNG wire#w1
   // the same network as SCL:
   #"AV-61.04"(LOCK := #"lock 4",   // "Valve"
               LIOP_SEL := #init,
               L_AUT := #init,
               L_REMOTE := #init,
               L_RESET := #reset,
               AUT_OP := "BFT-61".Out_AV_CIP_Tank,
               L_MON := #init,
               INSTANCE := 'AV-61.04',
               QCMD_OP => "AV-61.04");
END_REGION

REGION Network 25: AV-61.05
   RUNG wire#powerrail
      #"AV-61.05"(AUT_OP := wire#w1, LOCK := #"lock 4", ERR_EXTERN :=, LIOP_SEL := #init, L_AUT := #init, L_REMOTE := #init, L_SIM :=, L_RESET := #reset, MAN_OP :=, SIM_OP :=, FB_OPEN :=, FB_CLOSE :=, L_MON := #init, MON_T :=, MON_T_CLOSE :=, INSTANCE := 'AV-61.05', RESTART :=, VISIBILITY :=, OPdwCmd :=, QdwState =>, QwState =>, QCLOSING =>, QCLOSE =>, QOPENING =>, QOPEN =>, QCMD_OP => "AV-61.05", QMON =>, QMON_ERR =>, QMON_T =>, QMON_T_CLOSE =>, QMAN_AUT =>, QREMOTE =>, QSIM =>, QLOCK =>, QERR =>, QERR_EXT =>, QwAlarm =>)
   END_RUNG
   RUNG wire#powerrail
      Contact( "BFT-61".Out_AV_CIP_Tank )
   END_RUNG wire#w1
   // the same network as SCL:
   #"AV-61.05"(LOCK := #"lock 4",   // "Valve"
               LIOP_SEL := #init,
               L_AUT := #init,
               L_REMOTE := #init,
               L_RESET := #reset,
               AUT_OP := "BFT-61".Out_AV_CIP_Tank,
               L_MON := #init,
               INSTANCE := 'AV-61.05',
               QCMD_OP => "AV-61.05");
END_REGION

REGION Network 26: AV-61.21
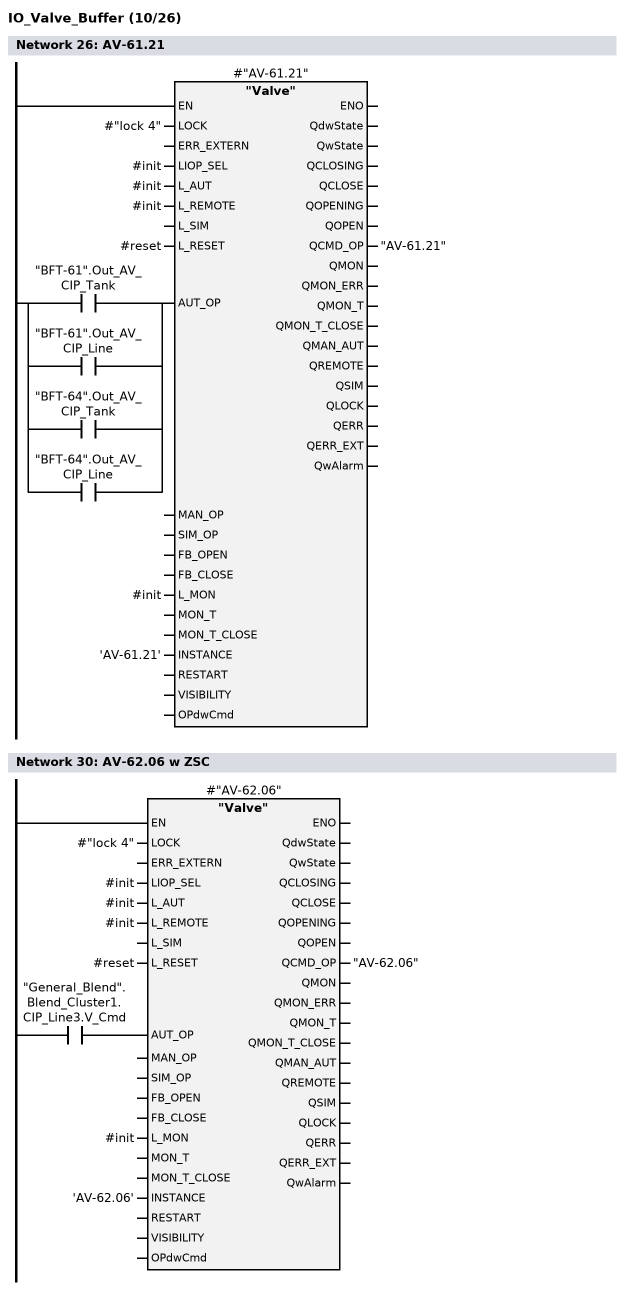
   RUNG wire#powerrail
      #"AV-61.21"(AUT_OP := wire#w1, LOCK := #"lock 4", ERR_EXTERN :=, LIOP_SEL := #init, L_AUT := #init, L_REMOTE := #init, L_SIM :=, L_RESET := #reset, MAN_OP :=, SIM_OP :=, FB_OPEN :=, FB_CLOSE :=, L_MON := #init, MON_T :=, MON_T_CLOSE :=, INSTANCE := 'AV-61.21', RESTART :=, VISIBILITY :=, OPdwCmd :=, QdwState =>, QwState =>, QCLOSING =>, QCLOSE =>, QOPENING =>, QOPEN =>, QCMD_OP => "AV-61.21", QMON =>, QMON_ERR =>, QMON_T =>, QMON_T_CLOSE =>, QMAN_AUT =>, QREMOTE =>, QSIM =>, QLOCK =>, QERR =>, QERR_EXT =>, QwAlarm =>)
   END_RUNG
   RUNG wire#powerrail
      Contact( "BFT-61".Out_AV_CIP_Tank )
   END_RUNG wire#w1
   RUNG wire#powerrail
      Contact( "BFT-61".Out_AV_CIP_Line )
   END_RUNG wire#w1
   RUNG wire#powerrail
      Contact( "BFT-64".Out_AV_CIP_Tank )
   END_RUNG wire#w1
   RUNG wire#powerrail
      Contact( "BFT-64".Out_AV_CIP_Line )
   END_RUNG wire#w1
   // the same network as SCL:
   #"AV-61.21"(LOCK := #"lock 4",   // "Valve"
               LIOP_SEL := #init,
               L_AUT := #init,
               L_REMOTE := #init,
               L_RESET := #reset,
               AUT_OP := "BFT-61".Out_AV_CIP_Tank OR "BFT-61".Out_AV_CIP_Line OR "BFT-64".Out_AV_CIP_Tank OR "BFT-64".Out_AV_CIP_Line,
               L_MON := #init,
               INSTANCE := 'AV-61.21',
               QCMD_OP => "AV-61.21");
END_REGION

REGION Network 28 (SCL): FB OPEN AND CLOSE VALVE T-62
   IF #testing THEN
       // Statement section IF
       #"AV-62.06".FB_OPEN := #"AV-62.06".QCMD_OP;
       #"AV-62.06".FB_CLOSE := NOT #"AV-62.06".QCMD_OP;
   ELSE
       // Statement section ELSE
       #"AV-62.06".FB_OPEN := NOT "ZSC-62.06";
       #"AV-62.06".FB_CLOSE := "ZSC-62.06";
   END_IF;
END_REGION

NETWORK
TITLE = FB MONITORING TIME VALVE T-62
// FB OPEN TIME
      L     T#20s;
      T     #"AV-62.06".MON_T;
// FB CLOSE TIME
      L     T#20s;
      T     #"AV-62.06".MON_T_CLOSE;

REGION Network 30: AV-62.06 w ZSC
   RUNG wire#powerrail
      #"AV-62.06"(AUT_OP := wire#w1, LOCK := #"lock 4", ERR_EXTERN :=, LIOP_SEL := #init, L_AUT := #init, L_REMOTE := #init, L_SIM :=, L_RESET := #reset, MAN_OP :=, SIM_OP :=, FB_OPEN :=, FB_CLOSE :=, L_MON := #init, MON_T :=, MON_T_CLOSE :=, INSTANCE := 'AV-62.06', RESTART :=, VISIBILITY :=, OPdwCmd :=, QdwState =>, QwState =>, QCLOSING =>, QCLOSE =>, QOPENING =>, QOPEN =>, QCMD_OP => "AV-62.06", QMON =>, QMON_ERR =>, QMON_T =>, QMON_T_CLOSE =>, QMAN_AUT =>, QREMOTE =>, QSIM =>, QLOCK =>, QERR =>, QERR_EXT =>, QwAlarm =>)
   END_RUNG
   RUNG wire#powerrail
      Contact( "General_Blend".Blend_Cluster1.CIP_Line3.V_Cmd )
   END_RUNG wire#w1
   // the same network as SCL:
   #"AV-62.06"(LOCK := #"lock 4",   // "Valve"
               LIOP_SEL := #init,
               L_AUT := #init,
               L_REMOTE := #init,
               L_RESET := #reset,
               AUT_OP := "General_Blend".Blend_Cluster1.CIP_Line3.V_Cmd,
               L_MON := #init,
               INSTANCE := 'AV-62.06',
               QCMD_OP => "AV-62.06");
END_REGION

REGION Network 32 (SCL): FB OPEN AND CLOSE VALVE T-64
   IF #testing THEN
       // Statement section IF
       #"AV-64.01".FB_OPEN := #"AV-64.01".QCMD_OP;
       #"AV-64.01".FB_CLOSE := NOT #"AV-64.01".QCMD_OP;
       #"AV-64.02".FB_OPEN := #"AV-64.02".QCMD_OP;
       #"AV-64.02".FB_CLOSE := NOT #"AV-64.02".QCMD_OP;
       #"AV-64.03".FB_OPEN := #"AV-64.03".QCMD_OP;
       #"AV-64.03".FB_CLOSE := NOT #"AV-64.03".QCMD_OP;
       #"AV-64.04".FB_OPEN := #"AV-64.04".QCMD_OP;
       #"AV-64.04".FB_CLOSE := NOT #"AV-64.04".QCMD_OP;
       #"AV-64.05".FB_OPEN := #"AV-64.05".QCMD_OP;
       #"AV-64.05".FB_CLOSE := NOT #"AV-64.05".QCMD_OP;
       #"AV-64.06".FB_OPEN := #"AV-64.06".QCMD_OP;
       #"AV-64.06".FB_CLOSE := NOT #"AV-64.06".QCMD_OP;
   ELSE
       // Statement section ELSE
       #"AV-64.01".FB_OPEN := NOT "ZSC-64.01";
       #"AV-64.01".FB_CLOSE := "ZSC-64.01";
       #"AV-64.02".FB_OPEN := #"AV-64.02".QCMD_OP;
       #"AV-64.02".FB_CLOSE := NOT #"AV-64.02".QCMD_OP;
       #"AV-64.03".FB_OPEN := NOT "ZSC-64.03";
       #"AV-64.03".FB_CLOSE := "ZSC-64.03";
       #"AV-64.04".FB_OPEN := #"AV-64.04".QCMD_OP;
       #"AV-64.04".FB_CLOSE := NOT #"AV-64.04".QCMD_OP;
       #"AV-64.05".FB_OPEN := #"AV-64.05".QCMD_OP;
       #"AV-64.05".FB_CLOSE := NOT #"AV-64.05".QCMD_OP;
       #"AV-64.06".FB_OPEN := NOT "ZSC-64.06";
       #"AV-64.06".FB_CLOSE := "ZSC-64.06";

   END_IF;
END_REGION

NETWORK
TITLE = FB MONITORING TIME VALVE T-64
// FB OPEN TIME
      L     T#20s;
      T     #"AV-64.01".MON_T;
      T     #"AV-64.02".MON_T;
      T     #"AV-64.03".MON_T;
      T     #"AV-64.04".MON_T;
      T     #"AV-64.05".MON_T;
      T     #"AV-64.06".MON_T;
// FB CLOSE TIME
      L     T#20s;
      T     #"AV-64.01".MON_T_CLOSE;
      T     #"AV-64.02".MON_T_CLOSE;
      T     #"AV-64.03".MON_T_CLOSE;
      T     #"AV-64.04".MON_T_CLOSE;
      T     #"AV-64.05".MON_T_CLOSE;
      T     #"AV-64.06".MON_T_CLOSE;

REGION Network 34: AV-64.01 w ZSC
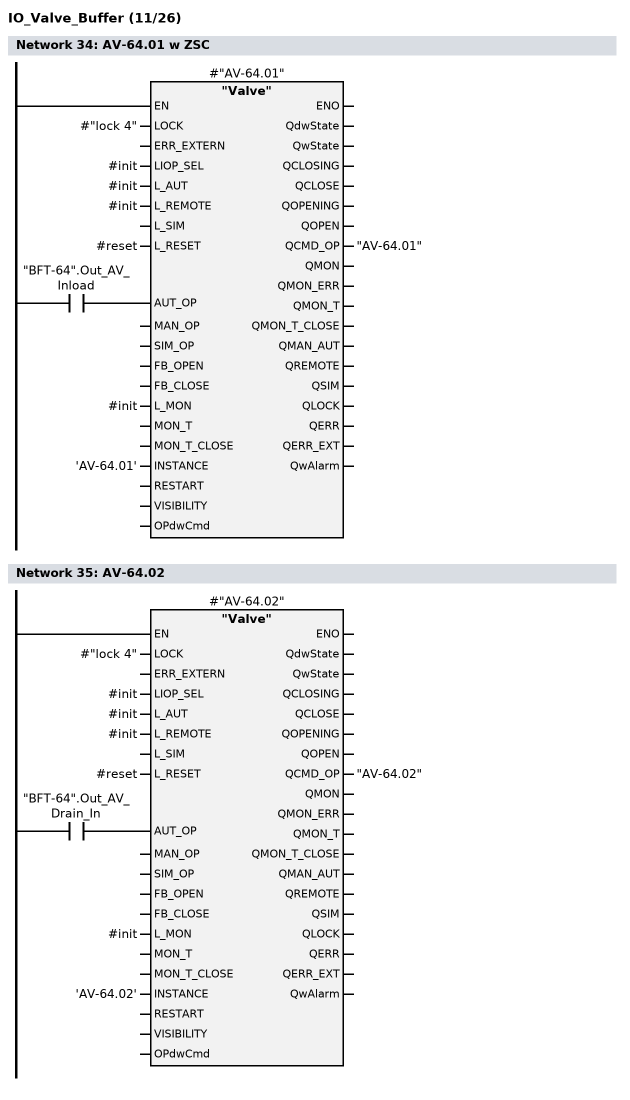
   RUNG wire#powerrail
      #"AV-64.01"(AUT_OP := wire#w1, LOCK := #"lock 4", ERR_EXTERN :=, LIOP_SEL := #init, L_AUT := #init, L_REMOTE := #init, L_SIM :=, L_RESET := #reset, MAN_OP :=, SIM_OP :=, FB_OPEN :=, FB_CLOSE :=, L_MON := #init, MON_T :=, MON_T_CLOSE :=, INSTANCE := 'AV-64.01', RESTART :=, VISIBILITY :=, OPdwCmd :=, QdwState =>, QwState =>, QCLOSING =>, QCLOSE =>, QOPENING =>, QOPEN =>, QCMD_OP => "AV-64.01", QMON =>, QMON_ERR =>, QMON_T =>, QMON_T_CLOSE =>, QMAN_AUT =>, QREMOTE =>, QSIM =>, QLOCK =>, QERR =>, QERR_EXT =>, QwAlarm =>)
   END_RUNG
   RUNG wire#powerrail
      Contact( "BFT-64".Out_AV_Inload )
   END_RUNG wire#w1
   // the same network as SCL:
   #"AV-64.01"(LOCK := #"lock 4",   // "Valve"
               LIOP_SEL := #init,
               L_AUT := #init,
               L_REMOTE := #init,
               L_RESET := #reset,
               AUT_OP := "BFT-64".Out_AV_Inload,
               L_MON := #init,
               INSTANCE := 'AV-64.01',
               QCMD_OP => "AV-64.01");
END_REGION

REGION Network 35: AV-64.02
   RUNG wire#powerrail
      #"AV-64.02"(AUT_OP := wire#w1, LOCK := #"lock 4", ERR_EXTERN :=, LIOP_SEL := #init, L_AUT := #init, L_REMOTE := #init, L_SIM :=, L_RESET := #reset, MAN_OP :=, SIM_OP :=, FB_OPEN :=, FB_CLOSE :=, L_MON := #init, MON_T :=, MON_T_CLOSE :=, INSTANCE := 'AV-64.02', RESTART :=, VISIBILITY :=, OPdwCmd :=, QdwState =>, QwState =>, QCLOSING =>, QCLOSE =>, QOPENING =>, QOPEN =>, QCMD_OP => "AV-64.02", QMON =>, QMON_ERR =>, QMON_T =>, QMON_T_CLOSE =>, QMAN_AUT =>, QREMOTE =>, QSIM =>, QLOCK =>, QERR =>, QERR_EXT =>, QwAlarm =>)
   END_RUNG
   RUNG wire#powerrail
      Contact( "BFT-64".Out_AV_Drain_In )
   END_RUNG wire#w1
   // the same network as SCL:
   #"AV-64.02"(LOCK := #"lock 4",   // "Valve"
               LIOP_SEL := #init,
               L_AUT := #init,
               L_REMOTE := #init,
               L_RESET := #reset,
               AUT_OP := "BFT-64".Out_AV_Drain_In,
               L_MON := #init,
               INSTANCE := 'AV-64.02',
               QCMD_OP => "AV-64.02");
END_REGION

REGION Network 36: AV-64.03 w ZSC
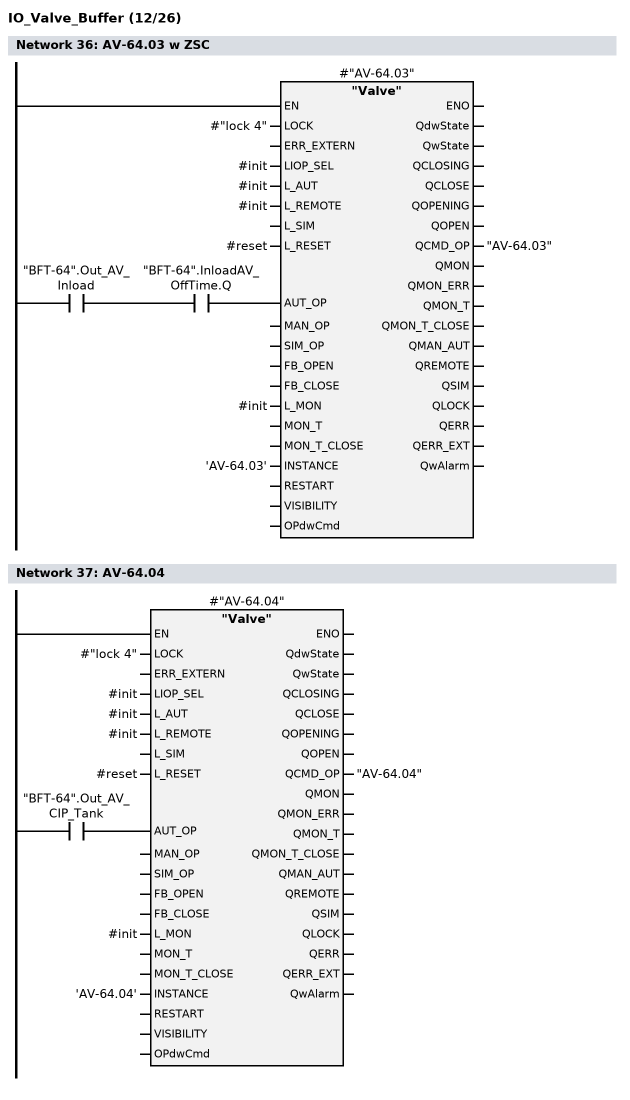
   RUNG wire#powerrail
      #"AV-64.03"(AUT_OP := wire#w1, LOCK := #"lock 4", ERR_EXTERN :=, LIOP_SEL := #init, L_AUT := #init, L_REMOTE := #init, L_SIM :=, L_RESET := #reset, MAN_OP :=, SIM_OP :=, FB_OPEN :=, FB_CLOSE :=, L_MON := #init, MON_T :=, MON_T_CLOSE :=, INSTANCE := 'AV-64.03', RESTART :=, VISIBILITY :=, OPdwCmd :=, QdwState =>, QwState =>, QCLOSING =>, QCLOSE =>, QOPENING =>, QOPEN =>, QCMD_OP => "AV-64.03", QMON =>, QMON_ERR =>, QMON_T =>, QMON_T_CLOSE =>, QMAN_AUT =>, QREMOTE =>, QSIM =>, QLOCK =>, QERR =>, QERR_EXT =>, QwAlarm =>)
   END_RUNG
   RUNG wire#powerrail
      Contact( "BFT-64".Out_AV_Inload )
      Contact( "BFT-64".InloadAV_OffTime.Q )
   END_RUNG wire#w1
   // the same network as SCL:
   #"AV-64.03"(LOCK := #"lock 4",   // "Valve"
               LIOP_SEL := #init,
               L_AUT := #init,
               L_REMOTE := #init,
               L_RESET := #reset,
               AUT_OP := "BFT-64".Out_AV_Inload AND "BFT-64".InloadAV_OffTime.Q,
               L_MON := #init,
               INSTANCE := 'AV-64.03',
               QCMD_OP => "AV-64.03");
END_REGION

REGION Network 37: AV-64.04
   RUNG wire#powerrail
      #"AV-64.04"(AUT_OP := wire#w1, LOCK := #"lock 4", ERR_EXTERN :=, LIOP_SEL := #init, L_AUT := #init, L_REMOTE := #init, L_SIM :=, L_RESET := #reset, MAN_OP :=, SIM_OP :=, FB_OPEN :=, FB_CLOSE :=, L_MON := #init, MON_T :=, MON_T_CLOSE :=, INSTANCE := 'AV-64.04', RESTART :=, VISIBILITY :=, OPdwCmd :=, QdwState =>, QwState =>, QCLOSING =>, QCLOSE =>, QOPENING =>, QOPEN =>, QCMD_OP => "AV-64.04", QMON =>, QMON_ERR =>, QMON_T =>, QMON_T_CLOSE =>, QMAN_AUT =>, QREMOTE =>, QSIM =>, QLOCK =>, QERR =>, QERR_EXT =>, QwAlarm =>)
   END_RUNG
   RUNG wire#powerrail
      Contact( "BFT-64".Out_AV_CIP_Tank )
   END_RUNG wire#w1
   // the same network as SCL:
   #"AV-64.04"(LOCK := #"lock 4",   // "Valve"
               LIOP_SEL := #init,
               L_AUT := #init,
               L_REMOTE := #init,
               L_RESET := #reset,
               AUT_OP := "BFT-64".Out_AV_CIP_Tank,
               L_MON := #init,
               INSTANCE := 'AV-64.04',
               QCMD_OP => "AV-64.04");
END_REGION

REGION Network 38: AV-64.05
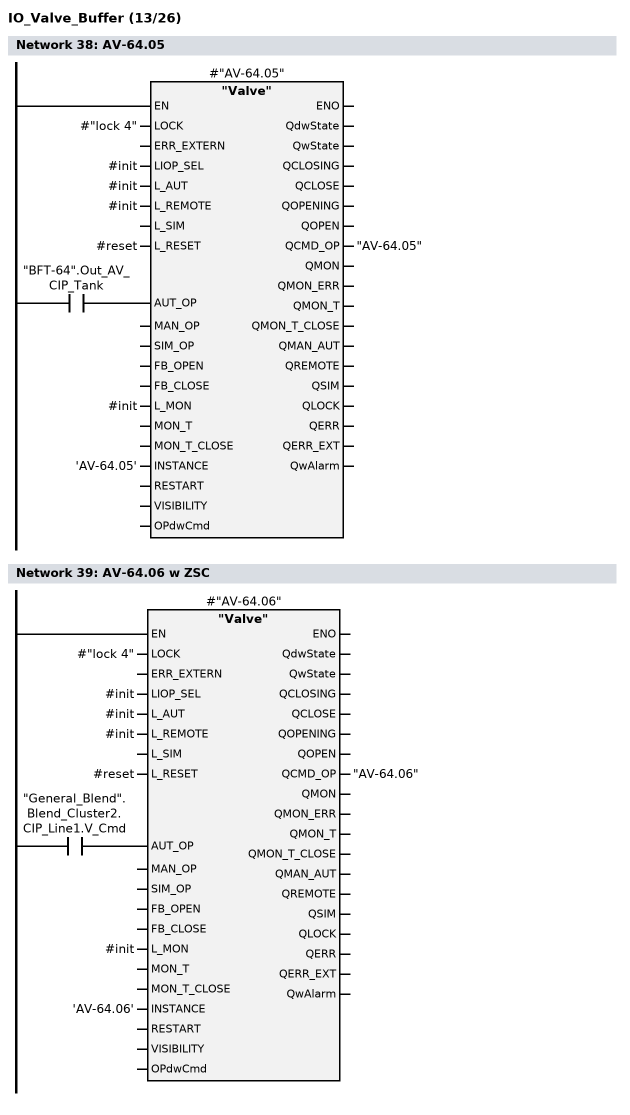
   RUNG wire#powerrail
      #"AV-64.05"(AUT_OP := wire#w1, LOCK := #"lock 4", ERR_EXTERN :=, LIOP_SEL := #init, L_AUT := #init, L_REMOTE := #init, L_SIM :=, L_RESET := #reset, MAN_OP :=, SIM_OP :=, FB_OPEN :=, FB_CLOSE :=, L_MON := #init, MON_T :=, MON_T_CLOSE :=, INSTANCE := 'AV-64.05', RESTART :=, VISIBILITY :=, OPdwCmd :=, QdwState =>, QwState =>, QCLOSING =>, QCLOSE =>, QOPENING =>, QOPEN =>, QCMD_OP => "AV-64.05", QMON =>, QMON_ERR =>, QMON_T =>, QMON_T_CLOSE =>, QMAN_AUT =>, QREMOTE =>, QSIM =>, QLOCK =>, QERR =>, QERR_EXT =>, QwAlarm =>)
   END_RUNG
   RUNG wire#powerrail
      Contact( "BFT-64".Out_AV_CIP_Tank )
   END_RUNG wire#w1
   // the same network as SCL:
   #"AV-64.05"(LOCK := #"lock 4",   // "Valve"
               LIOP_SEL := #init,
               L_AUT := #init,
               L_REMOTE := #init,
               L_RESET := #reset,
               AUT_OP := "BFT-64".Out_AV_CIP_Tank,
               L_MON := #init,
               INSTANCE := 'AV-64.05',
               QCMD_OP => "AV-64.05");
END_REGION

REGION Network 39: AV-64.06 w ZSC
   RUNG wire#powerrail
      #"AV-64.06"(AUT_OP := wire#w1, LOCK := #"lock 4", ERR_EXTERN :=, LIOP_SEL := #init, L_AUT := #init, L_REMOTE := #init, L_SIM :=, L_RESET := #reset, MAN_OP :=, SIM_OP :=, FB_OPEN :=, FB_CLOSE :=, L_MON := #init, MON_T :=, MON_T_CLOSE :=, INSTANCE := 'AV-64.06', RESTART :=, VISIBILITY :=, OPdwCmd :=, QdwState =>, QwState =>, QCLOSING =>, QCLOSE =>, QOPENING =>, QOPEN =>, QCMD_OP => "AV-64.06", QMON =>, QMON_ERR =>, QMON_T =>, QMON_T_CLOSE =>, QMAN_AUT =>, QREMOTE =>, QSIM =>, QLOCK =>, QERR =>, QERR_EXT =>, QwAlarm =>)
   END_RUNG
   RUNG wire#powerrail
      Contact( "General_Blend".Blend_Cluster2.CIP_Line1.V_Cmd )
   END_RUNG wire#w1
   // the same network as SCL:
   #"AV-64.06"(LOCK := #"lock 4",   // "Valve"
               LIOP_SEL := #init,
               L_AUT := #init,
               L_REMOTE := #init,
               L_RESET := #reset,
               AUT_OP := "General_Blend".Blend_Cluster2.CIP_Line1.V_Cmd,
               L_MON := #init,
               INSTANCE := 'AV-64.06',
               QCMD_OP => "AV-64.06");
END_REGION

REGION Network 41 (SCL): FB OPEN AND CLOSE VALVE T-65
   IF #testing THEN
       // Statement section IF
       #"AV-65.01".FB_OPEN := #"AV-65.01".QCMD_OP;
       #"AV-65.01".FB_CLOSE := NOT #"AV-65.01".QCMD_OP;
       #"AV-65.02".FB_OPEN := #"AV-65.02".QCMD_OP;
       #"AV-65.02".FB_CLOSE := NOT #"AV-65.02".QCMD_OP;
       #"AV-65.03".FB_OPEN := #"AV-65.03".QCMD_OP;
       #"AV-65.03".FB_CLOSE := NOT #"AV-65.03".QCMD_OP;
       #"AV-65.04".FB_OPEN := #"AV-65.04".QCMD_OP;
       #"AV-65.04".FB_CLOSE := NOT #"AV-65.04".QCMD_OP;
       #"AV-65.05".FB_OPEN := #"AV-65.05".QCMD_OP;
       #"AV-65.05".FB_CLOSE := NOT #"AV-65.05".QCMD_OP;
       #"AV-65.21".FB_OPEN := #"AV-65.21".QCMD_OP;
       #"AV-65.21".FB_CLOSE := NOT #"AV-65.21".QCMD_OP;
   ELSE
       // Statement section ELSE
       #"AV-65.01".FB_OPEN := NOT "ZSC-65.01";
       #"AV-65.01".FB_CLOSE := "ZSC-65.01";
       #"AV-65.02".FB_OPEN := #"AV-65.02".QCMD_OP;
       #"AV-65.02".FB_CLOSE := NOT #"AV-65.02".QCMD_OP;
       #"AV-65.03".FB_OPEN := NOT "ZSC-65.03";
       #"AV-65.03".FB_CLOSE := "ZSC-65.03";
       #"AV-65.04".FB_OPEN := #"AV-65.04".QCMD_OP;
       #"AV-65.04".FB_CLOSE := NOT #"AV-65.04".QCMD_OP;
       #"AV-65.05".FB_OPEN := #"AV-65.05".QCMD_OP;
       #"AV-65.05".FB_CLOSE := NOT #"AV-65.05".QCMD_OP;
       #"AV-65.21".FB_OPEN := #"AV-65.21".QCMD_OP;
       #"AV-65.21".FB_CLOSE := NOT #"AV-65.21".QCMD_OP;
   END_IF;
END_REGION

NETWORK
TITLE = FB MONITORING TIME VALVE T-65
// FB OPEN TIME
      L     T#20s;
      T     #"AV-65.01".MON_T;
      T     #"AV-65.02".MON_T;
      T     #"AV-65.03".MON_T;
      T     #"AV-65.04".MON_T;
      T     #"AV-65.05".MON_T;
      T     #"AV-65.21".MON_T;
// FB CLOSE TIME
      L     T#20s;
      T     #"AV-65.01".MON_T_CLOSE;
      T     #"AV-65.02".MON_T_CLOSE;
      T     #"AV-65.03".MON_T_CLOSE;
      T     #"AV-65.04".MON_T_CLOSE;
      T     #"AV-65.05".MON_T_CLOSE;
      T     #"AV-65.21".MON_T_CLOSE;

REGION Network 43: AV-65.01 w ZSC
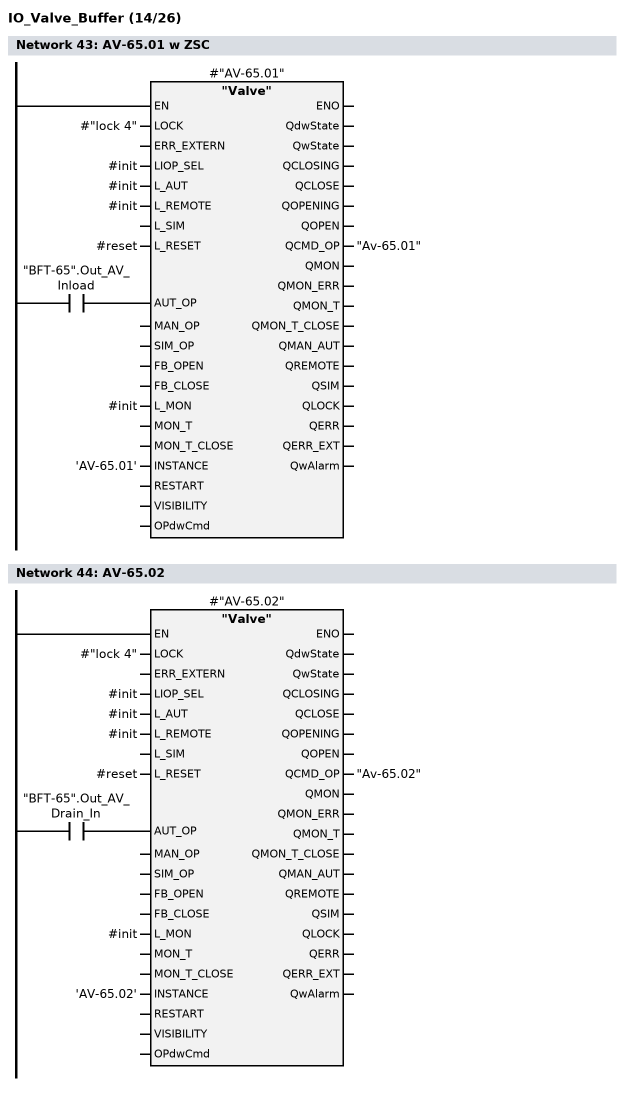
   RUNG wire#powerrail
      #"AV-65.01"(AUT_OP := wire#w1, LOCK := #"lock 4", ERR_EXTERN :=, LIOP_SEL := #init, L_AUT := #init, L_REMOTE := #init, L_SIM :=, L_RESET := #reset, MAN_OP :=, SIM_OP :=, FB_OPEN :=, FB_CLOSE :=, L_MON := #init, MON_T :=, MON_T_CLOSE :=, INSTANCE := 'AV-65.01', RESTART :=, VISIBILITY :=, OPdwCmd :=, QdwState =>, QwState =>, QCLOSING =>, QCLOSE =>, QOPENING =>, QOPEN =>, QCMD_OP => "Av-65.01", QMON =>, QMON_ERR =>, QMON_T =>, QMON_T_CLOSE =>, QMAN_AUT =>, QREMOTE =>, QSIM =>, QLOCK =>, QERR =>, QERR_EXT =>, QwAlarm =>)
   END_RUNG
   RUNG wire#powerrail
      Contact( "BFT-65".Out_AV_Inload )
   END_RUNG wire#w1
   // the same network as SCL:
   #"AV-65.01"(LOCK := #"lock 4",   // "Valve"
               LIOP_SEL := #init,
               L_AUT := #init,
               L_REMOTE := #init,
               L_RESET := #reset,
               AUT_OP := "BFT-65".Out_AV_Inload,
               L_MON := #init,
               INSTANCE := 'AV-65.01',
               QCMD_OP => "Av-65.01");
END_REGION

REGION Network 44: AV-65.02
   RUNG wire#powerrail
      #"AV-65.02"(AUT_OP := wire#w1, LOCK := #"lock 4", ERR_EXTERN :=, LIOP_SEL := #init, L_AUT := #init, L_REMOTE := #init, L_SIM :=, L_RESET := #reset, MAN_OP :=, SIM_OP :=, FB_OPEN :=, FB_CLOSE :=, L_MON := #init, MON_T :=, MON_T_CLOSE :=, INSTANCE := 'AV-65.02', RESTART :=, VISIBILITY :=, OPdwCmd :=, QdwState =>, QwState =>, QCLOSING =>, QCLOSE =>, QOPENING =>, QOPEN =>, QCMD_OP => "Av-65.02", QMON =>, QMON_ERR =>, QMON_T =>, QMON_T_CLOSE =>, QMAN_AUT =>, QREMOTE =>, QSIM =>, QLOCK =>, QERR =>, QERR_EXT =>, QwAlarm =>)
   END_RUNG
   RUNG wire#powerrail
      Contact( "BFT-65".Out_AV_Drain_In )
   END_RUNG wire#w1
   // the same network as SCL:
   #"AV-65.02"(LOCK := #"lock 4",   // "Valve"
               LIOP_SEL := #init,
               L_AUT := #init,
               L_REMOTE := #init,
               L_RESET := #reset,
               AUT_OP := "BFT-65".Out_AV_Drain_In,
               L_MON := #init,
               INSTANCE := 'AV-65.02',
               QCMD_OP => "Av-65.02");
END_REGION

REGION Network 45: AV-65.03 w ZSC
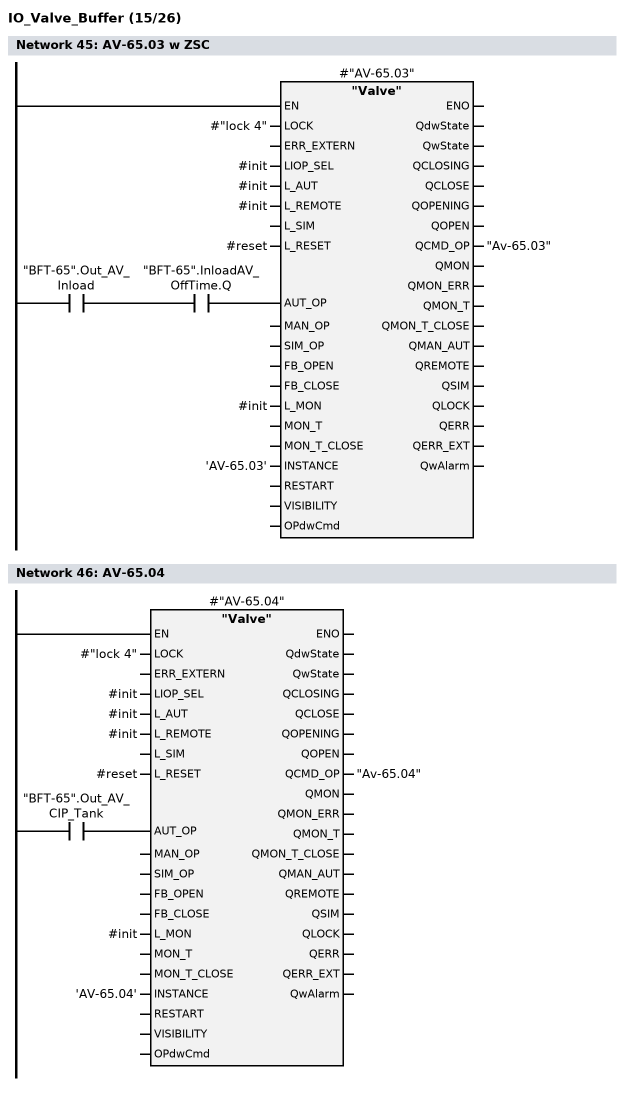
   RUNG wire#powerrail
      #"AV-65.03"(AUT_OP := wire#w1, LOCK := #"lock 4", ERR_EXTERN :=, LIOP_SEL := #init, L_AUT := #init, L_REMOTE := #init, L_SIM :=, L_RESET := #reset, MAN_OP :=, SIM_OP :=, FB_OPEN :=, FB_CLOSE :=, L_MON := #init, MON_T :=, MON_T_CLOSE :=, INSTANCE := 'AV-65.03', RESTART :=, VISIBILITY :=, OPdwCmd :=, QdwState =>, QwState =>, QCLOSING =>, QCLOSE =>, QOPENING =>, QOPEN =>, QCMD_OP => "Av-65.03", QMON =>, QMON_ERR =>, QMON_T =>, QMON_T_CLOSE =>, QMAN_AUT =>, QREMOTE =>, QSIM =>, QLOCK =>, QERR =>, QERR_EXT =>, QwAlarm =>)
   END_RUNG
   RUNG wire#powerrail
      Contact( "BFT-65".Out_AV_Inload )
      Contact( "BFT-65".InloadAV_OffTime.Q )
   END_RUNG wire#w1
   // the same network as SCL:
   #"AV-65.03"(LOCK := #"lock 4",   // "Valve"
               LIOP_SEL := #init,
               L_AUT := #init,
               L_REMOTE := #init,
               L_RESET := #reset,
               AUT_OP := "BFT-65".Out_AV_Inload AND "BFT-65".InloadAV_OffTime.Q,
               L_MON := #init,
               INSTANCE := 'AV-65.03',
               QCMD_OP => "Av-65.03");
END_REGION

REGION Network 46: AV-65.04
   RUNG wire#powerrail
      #"AV-65.04"(AUT_OP := wire#w1, LOCK := #"lock 4", ERR_EXTERN :=, LIOP_SEL := #init, L_AUT := #init, L_REMOTE := #init, L_SIM :=, L_RESET := #reset, MAN_OP :=, SIM_OP :=, FB_OPEN :=, FB_CLOSE :=, L_MON := #init, MON_T :=, MON_T_CLOSE :=, INSTANCE := 'AV-65.04', RESTART :=, VISIBILITY :=, OPdwCmd :=, QdwState =>, QwState =>, QCLOSING =>, QCLOSE =>, QOPENING =>, QOPEN =>, QCMD_OP => "Av-65.04", QMON =>, QMON_ERR =>, QMON_T =>, QMON_T_CLOSE =>, QMAN_AUT =>, QREMOTE =>, QSIM =>, QLOCK =>, QERR =>, QERR_EXT =>, QwAlarm =>)
   END_RUNG
   RUNG wire#powerrail
      Contact( "BFT-65".Out_AV_CIP_Tank )
   END_RUNG wire#w1
   // the same network as SCL:
   #"AV-65.04"(LOCK := #"lock 4",   // "Valve"
               LIOP_SEL := #init,
               L_AUT := #init,
               L_REMOTE := #init,
               L_RESET := #reset,
               AUT_OP := "BFT-65".Out_AV_CIP_Tank,
               L_MON := #init,
               INSTANCE := 'AV-65.04',
               QCMD_OP => "Av-65.04");
END_REGION

REGION Network 47: AV-65.05
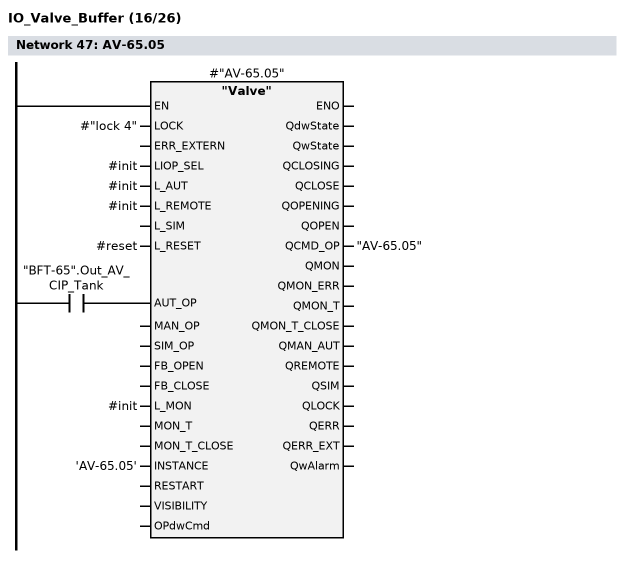
   RUNG wire#powerrail
      #"AV-65.05"(AUT_OP := wire#w1, LOCK := #"lock 4", ERR_EXTERN :=, LIOP_SEL := #init, L_AUT := #init, L_REMOTE := #init, L_SIM :=, L_RESET := #reset, MAN_OP :=, SIM_OP :=, FB_OPEN :=, FB_CLOSE :=, L_MON := #init, MON_T :=, MON_T_CLOSE :=, INSTANCE := 'AV-65.05', RESTART :=, VISIBILITY :=, OPdwCmd :=, QdwState =>, QwState =>, QCLOSING =>, QCLOSE =>, QOPENING =>, QOPEN =>, QCMD_OP => "AV-65.05", QMON =>, QMON_ERR =>, QMON_T =>, QMON_T_CLOSE =>, QMAN_AUT =>, QREMOTE =>, QSIM =>, QLOCK =>, QERR =>, QERR_EXT =>, QwAlarm =>)
   END_RUNG
   RUNG wire#powerrail
      Contact( "BFT-65".Out_AV_CIP_Tank )
   END_RUNG wire#w1
   // the same network as SCL:
   #"AV-65.05"(LOCK := #"lock 4",   // "Valve"
               LIOP_SEL := #init,
               L_AUT := #init,
               L_REMOTE := #init,
               L_RESET := #reset,
               AUT_OP := "BFT-65".Out_AV_CIP_Tank,
               L_MON := #init,
               INSTANCE := 'AV-65.05',
               QCMD_OP => "AV-65.05");
END_REGION

REGION Network 48: AV-65.21
